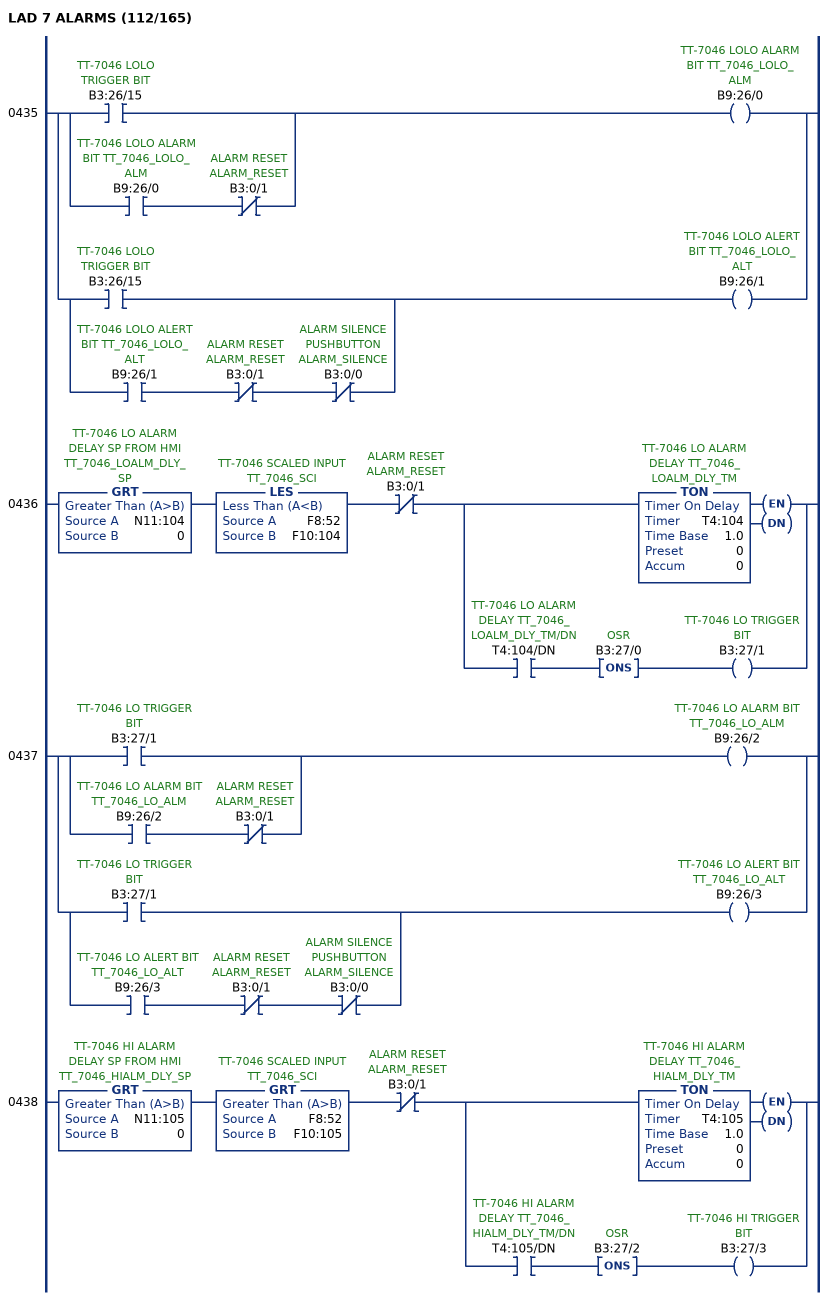
% Rung: 435 %
SOR BST BST XIC B3:26/15 NXB XIC B9:26/0 XIO B3:0/1 BND OTE B9:26/0 NXB BST XIC B3:26/15 NXB XIC B9:26/1 XIO B3:0/1 XIO B3:0/0 BND OTE B9:26/1 BND EOR
%   B3:26/15  "TT-7046 LOLO TRIGGER BIT" %
%   B9:26/0  TT_7046_LOLO_ALM  "TT-7046 LOLO ALARM BIT" %
%   B3:0/1  ALARM_RESET  "ALARM RESET" %
%   B9:26/1  TT_7046_LOLO_ALT  "TT-7046 LOLO ALERT BIT" %
%   B3:0/0  ALARM_SILENCE  "ALARM SILENCE PUSHBUTTON" %
% Rung: 436 %
SOR GRT N11:104 0 LES F8:52 F10:104 XIO B3:0/1 BST TON T4:104 1.0 0 0 NXB XIC T4:104/DN OSR B3:27/0 OTE B3:27/1 BND EOR
%   N11:104  TT_7046_LOALM_DLY_SP  "TT-7046 LO ALARM DELAY SP FROM HMI" %
%   F8:52  TT_7046_SCI  "TT-7046 SCALED INPUT" %
%   F10:104  TT_7046_LOALM_SP  "TT-7046 LO ALARM SP" %
%   B3:0/1  ALARM_RESET  "ALARM RESET" %
%   T4:104  TT_7046_LOALM_DLY_TM  "TT-7046 LO ALARM DELAY" %
%   B3:27/0  "OSR" %
%   B3:27/1  "TT-7046 LO TRIGGER BIT" %
% Rung: 437 %
SOR BST BST XIC B3:27/1 NXB XIC B9:26/2 XIO B3:0/1 BND OTE B9:26/2 NXB BST XIC B3:27/1 NXB XIC B9:26/3 XIO B3:0/1 XIO B3:0/0 BND OTE B9:26/3 BND EOR
%   B3:27/1  "TT-7046 LO TRIGGER BIT" %
%   B9:26/2  TT_7046_LO_ALM  "TT-7046 LO ALARM BIT" %
%   B3:0/1  ALARM_RESET  "ALARM RESET" %
%   B9:26/3  TT_7046_LO_ALT  "TT-7046 LO ALERT BIT" %
%   B3:0/0  ALARM_SILENCE  "ALARM SILENCE PUSHBUTTON" %
% Rung: 438 %
SOR GRT N11:105 0 GRT F8:52 F10:105 XIO B3:0/1 BST TON T4:105 1.0 0 0 NXB XIC T4:105/DN OSR B3:27/2 OTE B3:27/3 BND EOR
%   N11:105  TT_7046_HIALM_DLY_SP  "TT-7046 HI ALARM DELAY SP FROM HMI" %
%   F8:52  TT_7046_SCI  "TT-7046 SCALED INPUT" %
%   F10:105  TT_7046_HIALM_SP  "TT-7046 HI ALARM SP" %
%   B3:0/1  ALARM_RESET  "ALARM RESET" %
%   T4:105  TT_7046_HIALM_DLY_TM  "TT-7046 HI ALARM DELAY" %
%   B3:27/2  "OSR" %
%   B3:27/3  "TT-7046 HI TRIGGER BIT" %

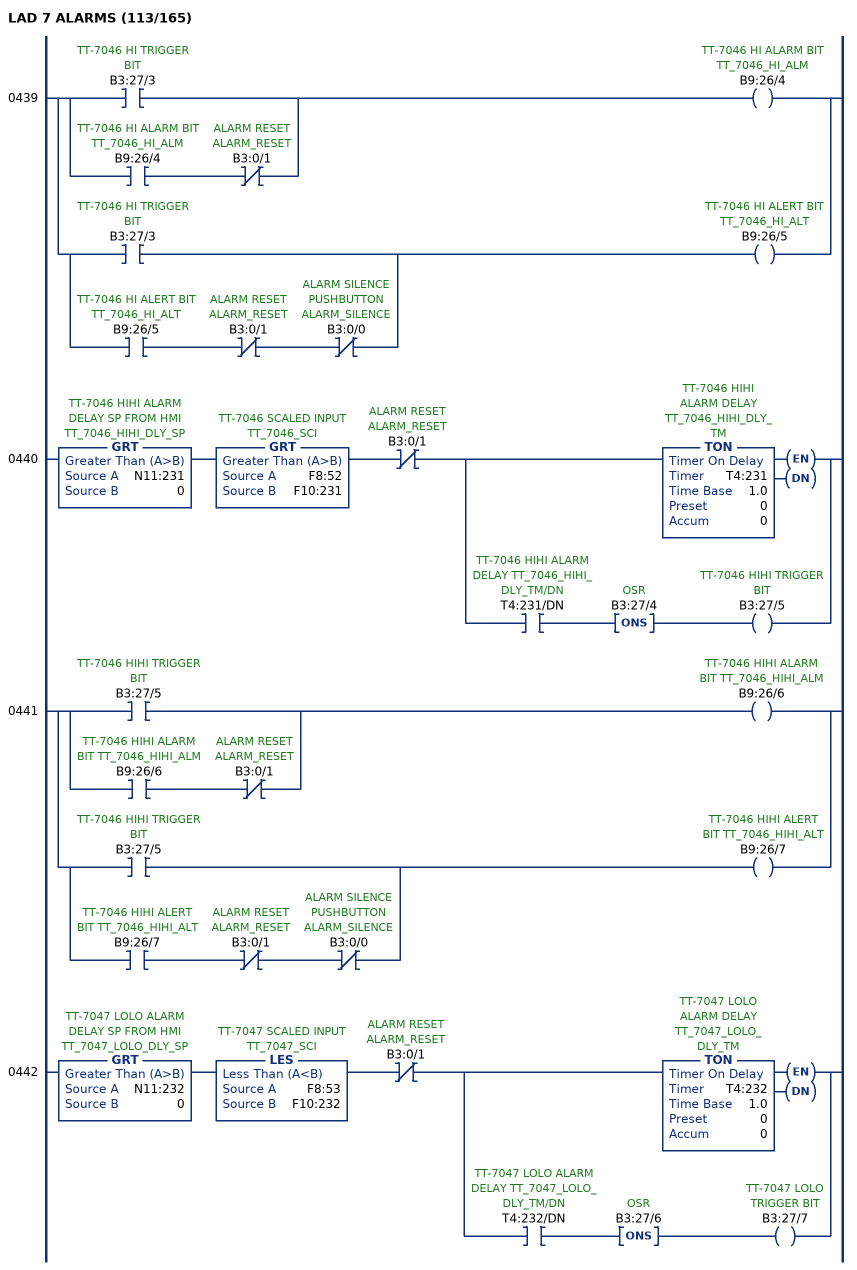
% Rung: 439 %
SOR BST BST XIC B3:27/3 NXB XIC B9:26/4 XIO B3:0/1 BND OTE B9:26/4 NXB BST XIC B3:27/3 NXB XIC B9:26/5 XIO B3:0/1 XIO B3:0/0 BND OTE B9:26/5 BND EOR
%   B3:27/3  "TT-7046 HI TRIGGER BIT" %
%   B9:26/4  TT_7046_HI_ALM  "TT-7046 HI ALARM BIT" %
%   B3:0/1  ALARM_RESET  "ALARM RESET" %
%   B9:26/5  TT_7046_HI_ALT  "TT-7046 HI ALERT BIT" %
%   B3:0/0  ALARM_SILENCE  "ALARM SILENCE PUSHBUTTON" %
% Rung: 440 %
SOR GRT N11:231 0 GRT F8:52 F10:231 XIO B3:0/1 BST TON T4:231 1.0 0 0 NXB XIC T4:231/DN OSR B3:27/4 OTE B3:27/5 BND EOR
%   N11:231  TT_7046_HIHI_DLY_SP  "TT-7046 HIHI ALARM DELAY SP FROM HMI" %
%   F8:52  TT_7046_SCI  "TT-7046 SCALED INPUT" %
%   F10:231  TT_7046_HIHI_SP  "TT-7046 HIHI ALARM SP" %
%   B3:0/1  ALARM_RESET  "ALARM RESET" %
%   T4:231  TT_7046_HIHI_DLY_TM  "TT-7046 HIHI ALARM DELAY" %
%   B3:27/4  "OSR" %
%   B3:27/5  "TT-7046 HIHI TRIGGER BIT" %
% Rung: 441 %
SOR BST BST XIC B3:27/5 NXB XIC B9:26/6 XIO B3:0/1 BND OTE B9:26/6 NXB BST XIC B3:27/5 NXB XIC B9:26/7 XIO B3:0/1 XIO B3:0/0 BND OTE B9:26/7 BND EOR
%   B3:27/5  "TT-7046 HIHI TRIGGER BIT" %
%   B9:26/6  TT_7046_HIHI_ALM  "TT-7046 HIHI ALARM BIT" %
%   B3:0/1  ALARM_RESET  "ALARM RESET" %
%   B9:26/7  TT_7046_HIHI_ALT  "TT-7046 HIHI ALERT BIT" %
%   B3:0/0  ALARM_SILENCE  "ALARM SILENCE PUSHBUTTON" %
% Rung: 442 %
SOR GRT N11:232 0 LES F8:53 F10:232 XIO B3:0/1 BST TON T4:232 1.0 0 0 NXB XIC T4:232/DN OSR B3:27/6 OTE B3:27/7 BND EOR
%   N11:232  TT_7047_LOLO_DLY_SP  "TT-7047 LOLO ALARM DELAY SP FROM HMI" %
%   F8:53  TT_7047_SCI  "TT-7047 SCALED INPUT" %
%   F10:232  TT_7047_LOLO_SP  "TT-7047 LOLO ALARM SP" %
%   B3:0/1  ALARM_RESET  "ALARM RESET" %
%   T4:232  TT_7047_LOLO_DLY_TM  "TT-7047 LOLO ALARM DELAY" %
%   B3:27/6  "OSR" %
%   B3:27/7  "TT-7047 LOLO TRIGGER BIT" %

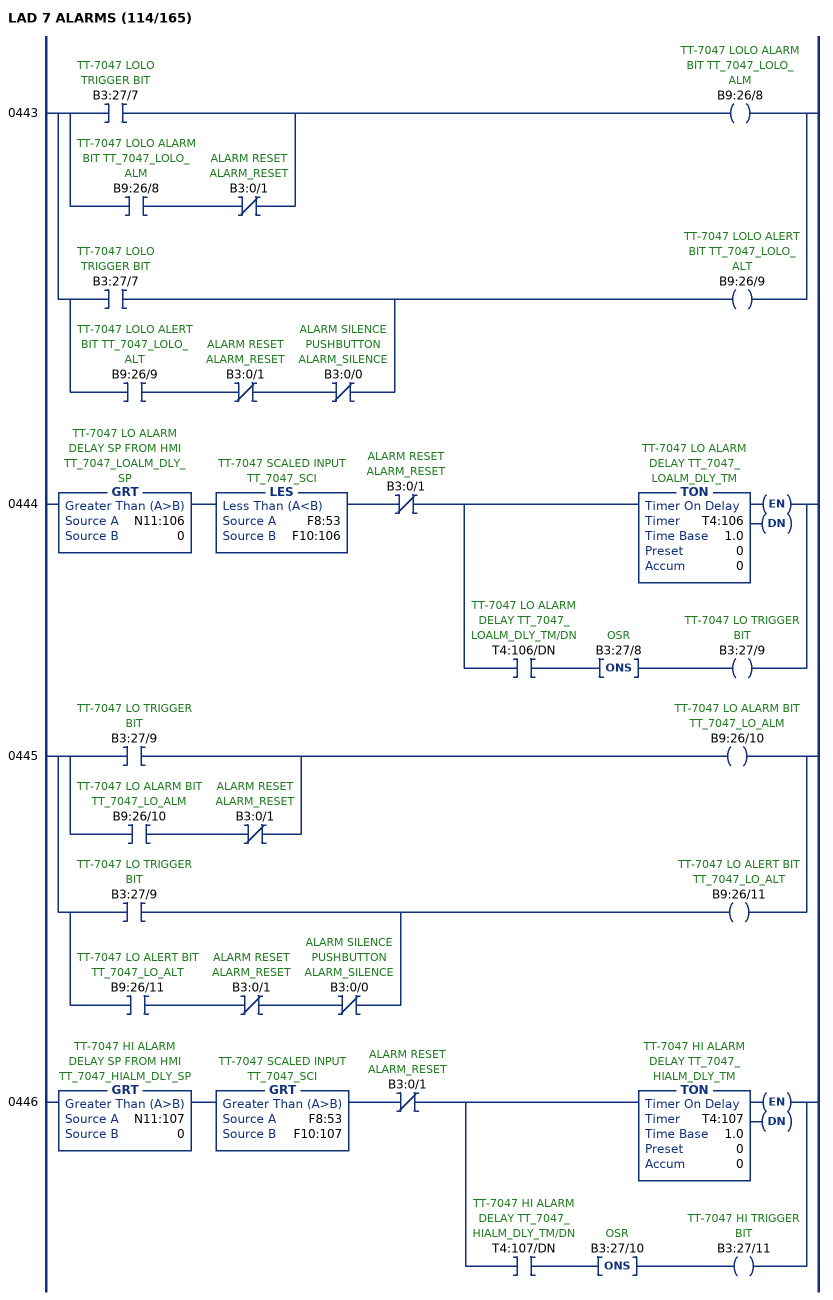
% Rung: 443 %
SOR BST BST XIC B3:27/7 NXB XIC B9:26/8 XIO B3:0/1 BND OTE B9:26/8 NXB BST XIC B3:27/7 NXB XIC B9:26/9 XIO B3:0/1 XIO B3:0/0 BND OTE B9:26/9 BND EOR
%   B3:27/7  "TT-7047 LOLO TRIGGER BIT" %
%   B9:26/8  TT_7047_LOLO_ALM  "TT-7047 LOLO ALARM BIT" %
%   B3:0/1  ALARM_RESET  "ALARM RESET" %
%   B9:26/9  TT_7047_LOLO_ALT  "TT-7047 LOLO ALERT BIT" %
%   B3:0/0  ALARM_SILENCE  "ALARM SILENCE PUSHBUTTON" %
% Rung: 444 %
SOR GRT N11:106 0 LES F8:53 F10:106 XIO B3:0/1 BST TON T4:106 1.0 0 0 NXB XIC T4:106/DN OSR B3:27/8 OTE B3:27/9 BND EOR
%   N11:106  TT_7047_LOALM_DLY_SP  "TT-7047 LO ALARM DELAY SP FROM HMI" %
%   F8:53  TT_7047_SCI  "TT-7047 SCALED INPUT" %
%   F10:106  TT_7047_LOALM_SP  "TT-7047 LO ALARM SP" %
%   B3:0/1  ALARM_RESET  "ALARM RESET" %
%   T4:106  TT_7047_LOALM_DLY_TM  "TT-7047 LO ALARM DELAY" %
%   B3:27/8  "OSR" %
%   B3:27/9  "TT-7047 LO TRIGGER BIT" %
% Rung: 445 %
SOR BST BST XIC B3:27/9 NXB XIC B9:26/10 XIO B3:0/1 BND OTE B9:26/10 NXB BST XIC B3:27/9 NXB XIC B9:26/11 XIO B3:0/1 XIO B3:0/0 BND OTE B9:26/11 BND EOR
%   B3:27/9  "TT-7047 LO TRIGGER BIT" %
%   B9:26/10  TT_7047_LO_ALM  "TT-7047 LO ALARM BIT" %
%   B3:0/1  ALARM_RESET  "ALARM RESET" %
%   B9:26/11  TT_7047_LO_ALT  "TT-7047 LO ALERT BIT" %
%   B3:0/0  ALARM_SILENCE  "ALARM SILENCE PUSHBUTTON" %
% Rung: 446 %
SOR GRT N11:107 0 GRT F8:53 F10:107 XIO B3:0/1 BST TON T4:107 1.0 0 0 NXB XIC T4:107/DN OSR B3:27/10 OTE B3:27/11 BND EOR
%   N11:107  TT_7047_HIALM_DLY_SP  "TT-7047 HI ALARM DELAY SP FROM HMI" %
%   F8:53  TT_7047_SCI  "TT-7047 SCALED INPUT" %
%   F10:107  TT_7047_HIALM_SP  "TT-7047 HI ALARM SP" %
%   B3:0/1  ALARM_RESET  "ALARM RESET" %
%   T4:107  TT_7047_HIALM_DLY_TM  "TT-7047 HI ALARM DELAY" %
%   B3:27/10  "OSR" %
%   B3:27/11  "TT-7047 HI TRIGGER BIT" %

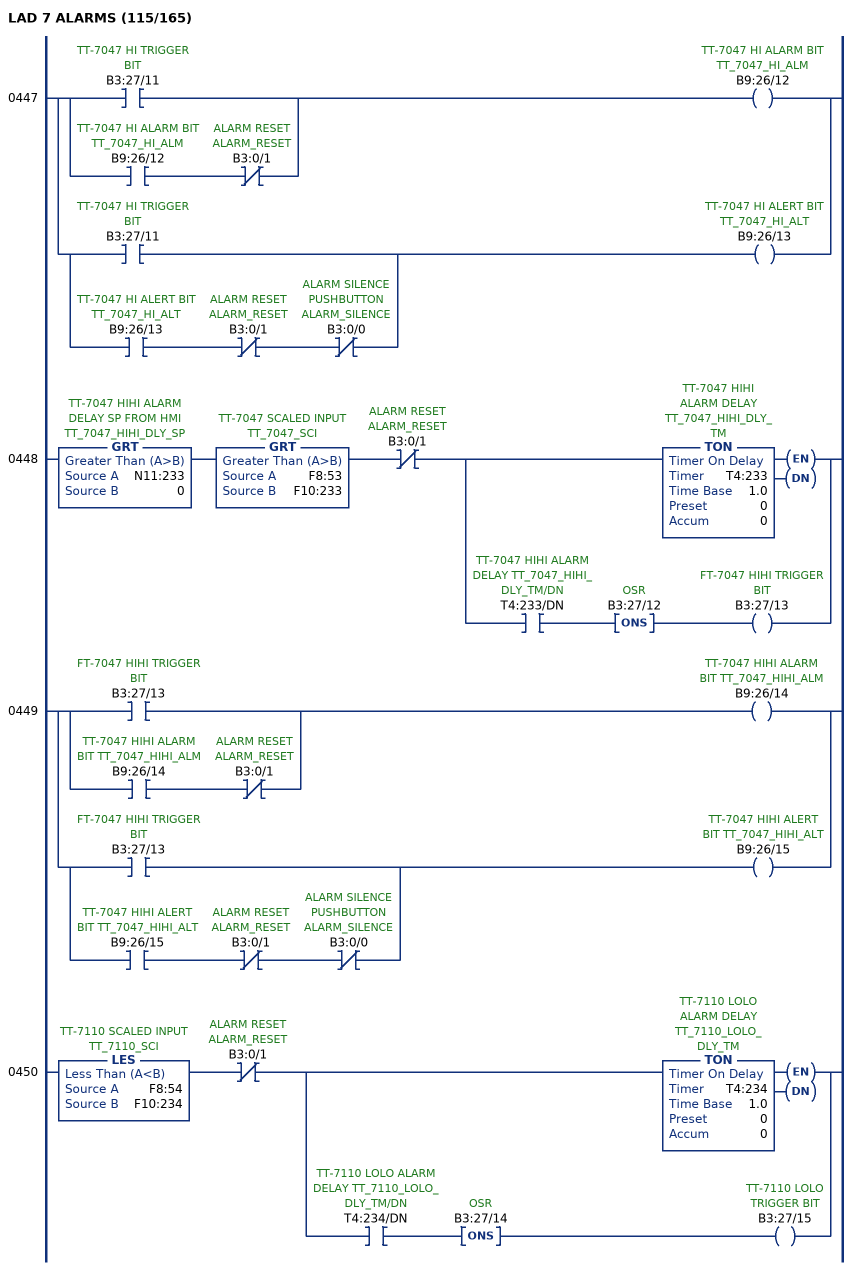
% Rung: 447 %
SOR BST BST XIC B3:27/11 NXB XIC B9:26/12 XIO B3:0/1 BND OTE B9:26/12 NXB BST XIC B3:27/11 NXB XIC B9:26/13 XIO B3:0/1 XIO B3:0/0 BND OTE B9:26/13 BND EOR
%   B3:27/11  "TT-7047 HI TRIGGER BIT" %
%   B9:26/12  TT_7047_HI_ALM  "TT-7047 HI ALARM BIT" %
%   B3:0/1  ALARM_RESET  "ALARM RESET" %
%   B9:26/13  TT_7047_HI_ALT  "TT-7047 HI ALERT BIT" %
%   B3:0/0  ALARM_SILENCE  "ALARM SILENCE PUSHBUTTON" %
% Rung: 448 %
SOR GRT N11:233 0 GRT F8:53 F10:233 XIO B3:0/1 BST TON T4:233 1.0 0 0 NXB XIC T4:233/DN OSR B3:27/12 OTE B3:27/13 BND EOR
%   N11:233  TT_7047_HIHI_DLY_SP  "TT-7047 HIHI ALARM DELAY SP FROM HMI" %
%   F8:53  TT_7047_SCI  "TT-7047 SCALED INPUT" %
%   F10:233  TT_7047_HIHI_SP  "TT-7047 HIHI ALARM SP" %
%   B3:0/1  ALARM_RESET  "ALARM RESET" %
%   T4:233  TT_7047_HIHI_DLY_TM  "TT-7047 HIHI ALARM DELAY" %
%   B3:27/12  "OSR" %
%   B3:27/13  "FT-7047 HIHI TRIGGER BIT" %
% Rung: 449 %
SOR BST BST XIC B3:27/13 NXB XIC B9:26/14 XIO B3:0/1 BND OTE B9:26/14 NXB BST XIC B3:27/13 NXB XIC B9:26/15 XIO B3:0/1 XIO B3:0/0 BND OTE B9:26/15 BND EOR
%   B3:27/13  "FT-7047 HIHI TRIGGER BIT" %
%   B9:26/14  TT_7047_HIHI_ALM  "TT-7047 HIHI ALARM BIT" %
%   B3:0/1  ALARM_RESET  "ALARM RESET" %
%   B9:26/15  TT_7047_HIHI_ALT  "TT-7047 HIHI ALERT BIT" %
%   B3:0/0  ALARM_SILENCE  "ALARM SILENCE PUSHBUTTON" %
% Rung: 450 %
SOR LES F8:54 F10:234 XIO B3:0/1 BST TON T4:234 1.0 0 0 NXB XIC T4:234/DN OSR B3:27/14 OTE B3:27/15 BND EOR
%   F8:54  TT_7110_SCI  "TT-7110 SCALED INPUT" %
%   F10:234  TT_7110_LOLO_SP  "TT-7110 LOLO ALARM SP" %
%   B3:0/1  ALARM_RESET  "ALARM RESET" %
%   T4:234  TT_7110_LOLO_DLY_TM  "TT-7110 LOLO ALARM DELAY" %
%   B3:27/14  "OSR" %
%   B3:27/15  "TT-7110 LOLO TRIGGER BIT" %

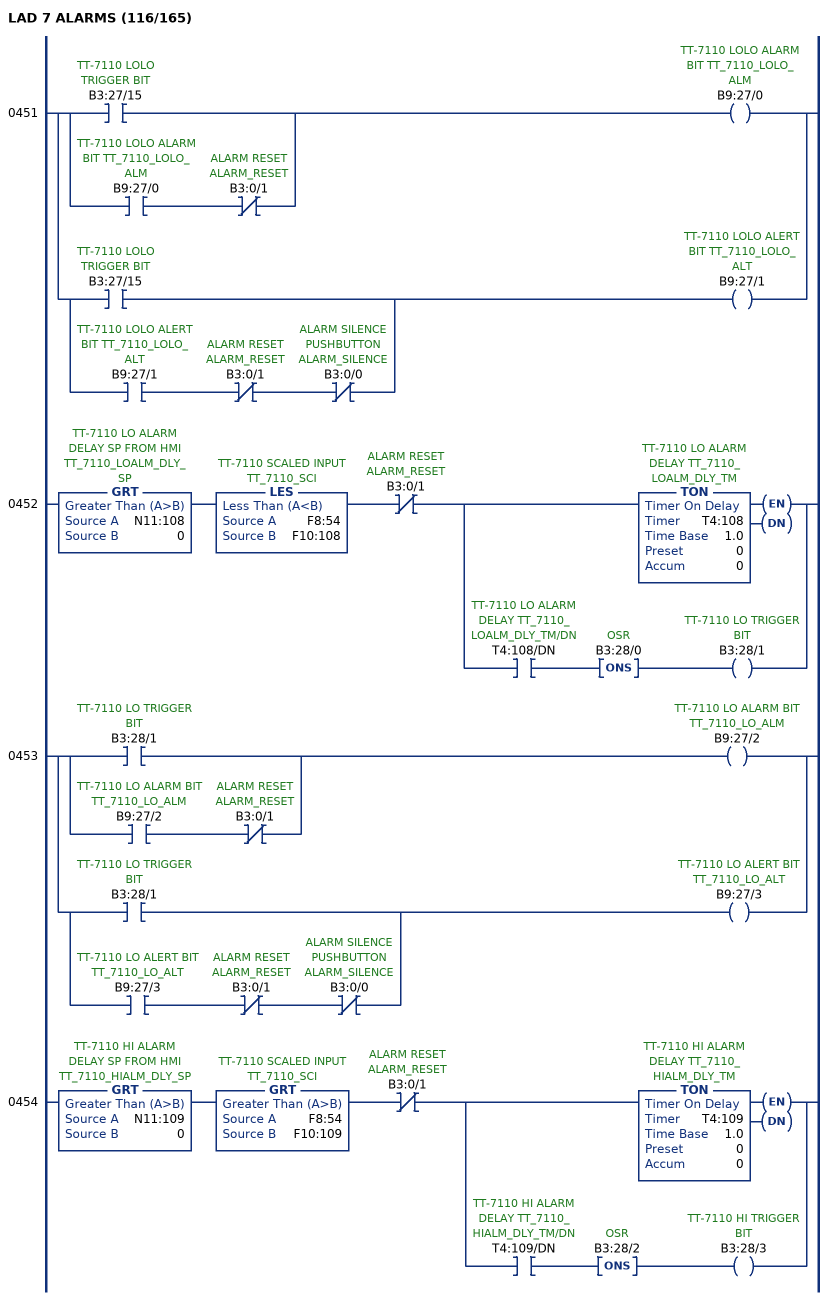
% Rung: 451 %
SOR BST BST XIC B3:27/15 NXB XIC B9:27/0 XIO B3:0/1 BND OTE B9:27/0 NXB BST XIC B3:27/15 NXB XIC B9:27/1 XIO B3:0/1 XIO B3:0/0 BND OTE B9:27/1 BND EOR
%   B3:27/15  "TT-7110 LOLO TRIGGER BIT" %
%   B9:27/0  TT_7110_LOLO_ALM  "TT-7110 LOLO ALARM BIT" %
%   B3:0/1  ALARM_RESET  "ALARM RESET" %
%   B9:27/1  TT_7110_LOLO_ALT  "TT-7110 LOLO ALERT BIT" %
%   B3:0/0  ALARM_SILENCE  "ALARM SILENCE PUSHBUTTON" %
% Rung: 452 %
SOR GRT N11:108 0 LES F8:54 F10:108 XIO B3:0/1 BST TON T4:108 1.0 0 0 NXB XIC T4:108/DN OSR B3:28/0 OTE B3:28/1 BND EOR
%   N11:108  TT_7110_LOALM_DLY_SP  "TT-7110 LO ALARM DELAY SP FROM HMI" %
%   F8:54  TT_7110_SCI  "TT-7110 SCALED INPUT" %
%   F10:108  TT_7110_LOALM_SP  "TT-7110 LO ALARM SP" %
%   B3:0/1  ALARM_RESET  "ALARM RESET" %
%   T4:108  TT_7110_LOALM_DLY_TM  "TT-7110 LO ALARM DELAY" %
%   B3:28/0  "OSR" %
%   B3:28/1  "TT-7110 LO TRIGGER BIT" %
% Rung: 453 %
SOR BST BST XIC B3:28/1 NXB XIC B9:27/2 XIO B3:0/1 BND OTE B9:27/2 NXB BST XIC B3:28/1 NXB XIC B9:27/3 XIO B3:0/1 XIO B3:0/0 BND OTE B9:27/3 BND EOR
%   B3:28/1  "TT-7110 LO TRIGGER BIT" %
%   B9:27/2  TT_7110_LO_ALM  "TT-7110 LO ALARM BIT" %
%   B3:0/1  ALARM_RESET  "ALARM RESET" %
%   B9:27/3  TT_7110_LO_ALT  "TT-7110 LO ALERT BIT" %
%   B3:0/0  ALARM_SILENCE  "ALARM SILENCE PUSHBUTTON" %
% Rung: 454 %
SOR GRT N11:109 0 GRT F8:54 F10:109 XIO B3:0/1 BST TON T4:109 1.0 0 0 NXB XIC T4:109/DN OSR B3:28/2 OTE B3:28/3 BND EOR
%   N11:109  TT_7110_HIALM_DLY_SP  "TT-7110 HI ALARM DELAY SP FROM HMI" %
%   F8:54  TT_7110_SCI  "TT-7110 SCALED INPUT" %
%   F10:109  TT_7110_HIALM_SP  "TT-7110 HI ALARM SP" %
%   B3:0/1  ALARM_RESET  "ALARM RESET" %
%   T4:109  TT_7110_HIALM_DLY_TM  "TT-7110 HI ALARM DELAY" %
%   B3:28/2  "OSR" %
%   B3:28/3  "TT-7110 HI TRIGGER BIT" %

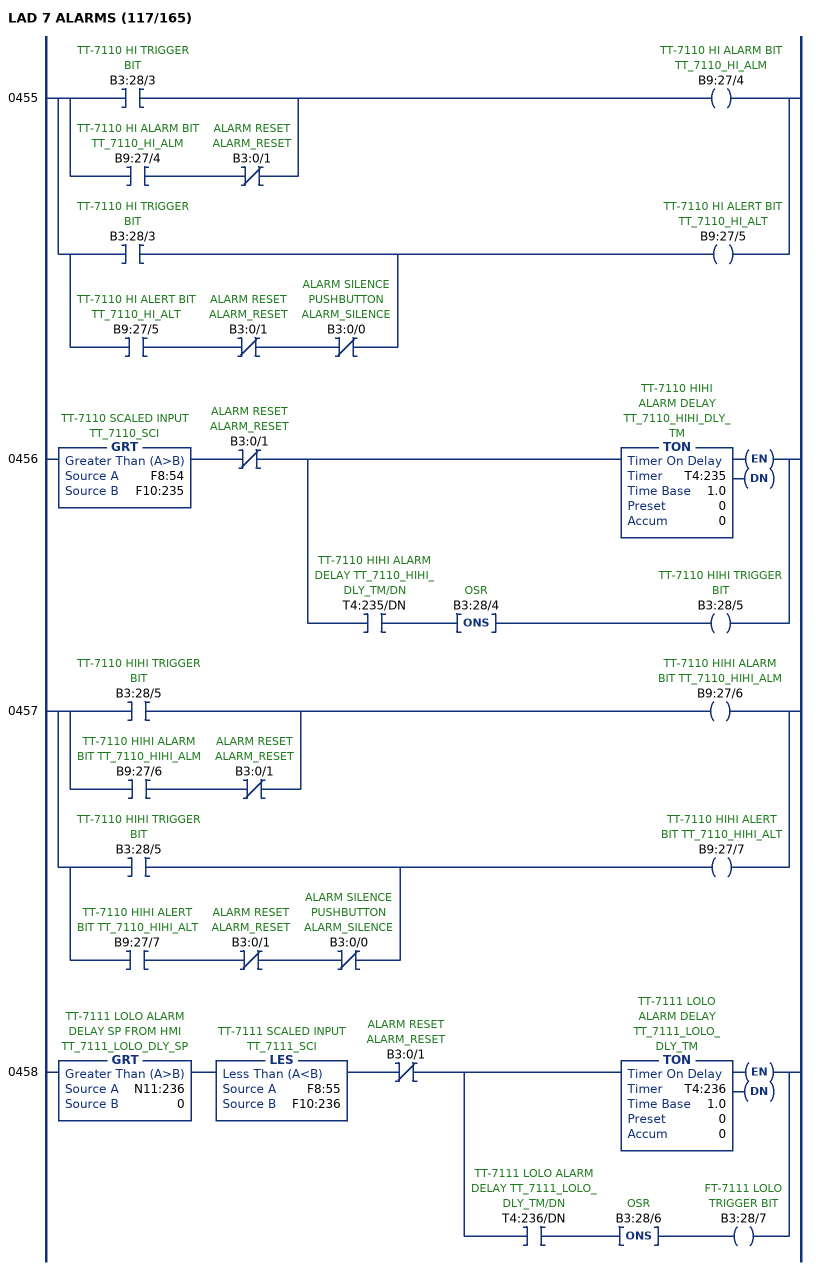
% Rung: 455 %
SOR BST BST XIC B3:28/3 NXB XIC B9:27/4 XIO B3:0/1 BND OTE B9:27/4 NXB BST XIC B3:28/3 NXB XIC B9:27/5 XIO B3:0/1 XIO B3:0/0 BND OTE B9:27/5 BND EOR
%   B3:28/3  "TT-7110 HI TRIGGER BIT" %
%   B9:27/4  TT_7110_HI_ALM  "TT-7110 HI ALARM BIT" %
%   B3:0/1  ALARM_RESET  "ALARM RESET" %
%   B9:27/5  TT_7110_HI_ALT  "TT-7110 HI ALERT BIT" %
%   B3:0/0  ALARM_SILENCE  "ALARM SILENCE PUSHBUTTON" %
% Rung: 456 %
SOR GRT F8:54 F10:235 XIO B3:0/1 BST TON T4:235 1.0 0 0 NXB XIC T4:235/DN OSR B3:28/4 OTE B3:28/5 BND EOR
%   F8:54  TT_7110_SCI  "TT-7110 SCALED INPUT" %
%   F10:235  TT_7110_HIHI_SP  "TT-7110 HIHI ALARM SP" %
%   B3:0/1  ALARM_RESET  "ALARM RESET" %
%   T4:235  TT_7110_HIHI_DLY_TM  "TT-7110 HIHI ALARM DELAY" %
%   B3:28/4  "OSR" %
%   B3:28/5  "TT-7110 HIHI TRIGGER BIT" %
% Rung: 457 %
SOR BST BST XIC B3:28/5 NXB XIC B9:27/6 XIO B3:0/1 BND OTE B9:27/6 NXB BST XIC B3:28/5 NXB XIC B9:27/7 XIO B3:0/1 XIO B3:0/0 BND OTE B9:27/7 BND EOR
%   B3:28/5  "TT-7110 HIHI TRIGGER BIT" %
%   B9:27/6  TT_7110_HIHI_ALM  "TT-7110 HIHI ALARM BIT" %
%   B3:0/1  ALARM_RESET  "ALARM RESET" %
%   B9:27/7  TT_7110_HIHI_ALT  "TT-7110 HIHI ALERT BIT" %
%   B3:0/0  ALARM_SILENCE  "ALARM SILENCE PUSHBUTTON" %
% Rung: 458 %
SOR GRT N11:236 0 LES F8:55 F10:236 XIO B3:0/1 BST TON T4:236 1.0 0 0 NXB XIC T4:236/DN OSR B3:28/6 OTE B3:28/7 BND EOR
%   N11:236  TT_7111_LOLO_DLY_SP  "TT-7111 LOLO ALARM DELAY SP FROM HMI" %
%   F8:55  TT_7111_SCI  "TT-7111 SCALED INPUT" %
%   F10:236  TT_7111_LOLO_SP  "TT-7111 LOLO ALARM SP" %
%   B3:0/1  ALARM_RESET  "ALARM RESET" %
%   T4:236  TT_7111_LOLO_DLY_TM  "TT-7111 LOLO ALARM DELAY" %
%   B3:28/6  "OSR" %
%   B3:28/7  "FT-7111 LOLO TRIGGER BIT" %

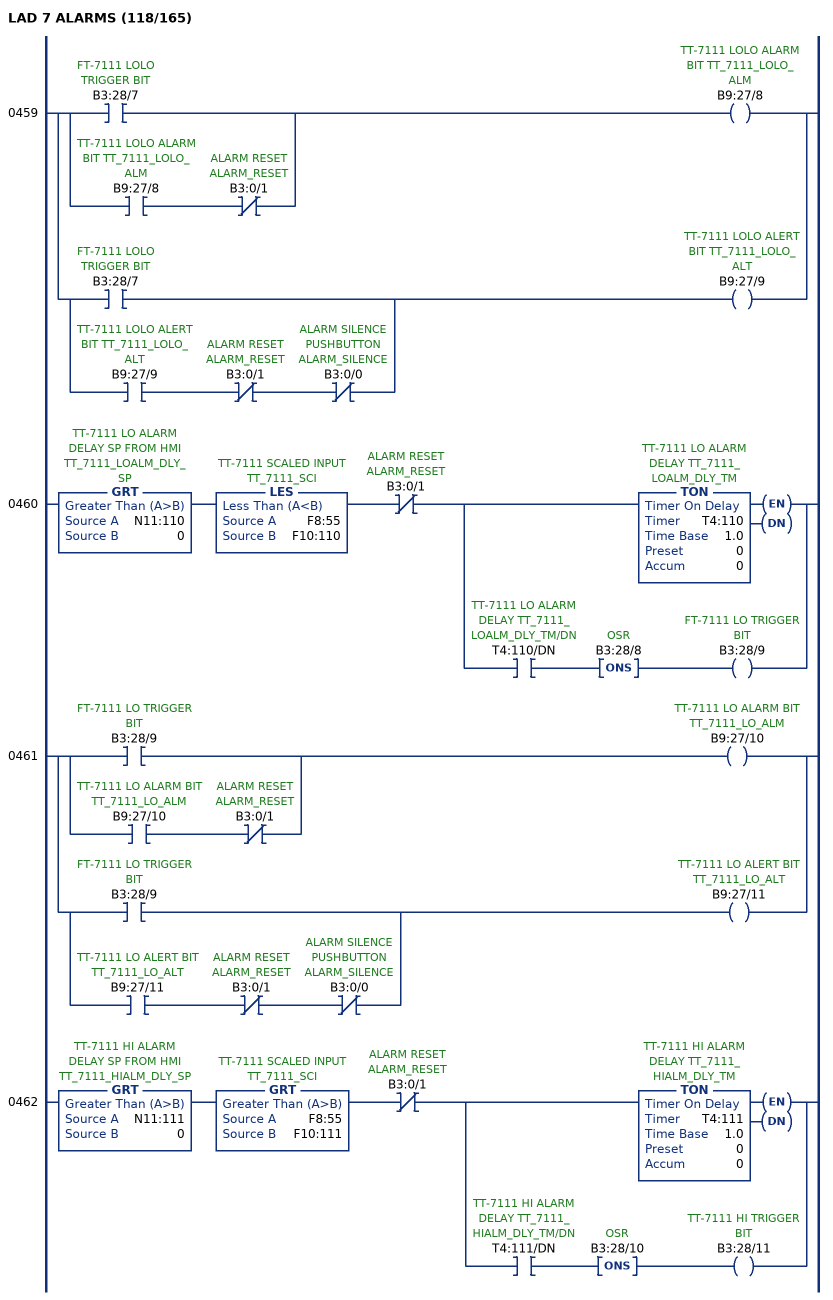
% Rung: 459 %
SOR BST BST XIC B3:28/7 NXB XIC B9:27/8 XIO B3:0/1 BND OTE B9:27/8 NXB BST XIC B3:28/7 NXB XIC B9:27/9 XIO B3:0/1 XIO B3:0/0 BND OTE B9:27/9 BND EOR
%   B3:28/7  "FT-7111 LOLO TRIGGER BIT" %
%   B9:27/8  TT_7111_LOLO_ALM  "TT-7111 LOLO ALARM BIT" %
%   B3:0/1  ALARM_RESET  "ALARM RESET" %
%   B9:27/9  TT_7111_LOLO_ALT  "TT-7111 LOLO ALERT BIT" %
%   B3:0/0  ALARM_SILENCE  "ALARM SILENCE PUSHBUTTON" %
% Rung: 460 %
SOR GRT N11:110 0 LES F8:55 F10:110 XIO B3:0/1 BST TON T4:110 1.0 0 0 NXB XIC T4:110/DN OSR B3:28/8 OTE B3:28/9 BND EOR
%   N11:110  TT_7111_LOALM_DLY_SP  "TT-7111 LO ALARM DELAY SP FROM HMI" %
%   F8:55  TT_7111_SCI  "TT-7111 SCALED INPUT" %
%   F10:110  TT_7111_LOALM_SP  "TT-7111 LO ALARM SP" %
%   B3:0/1  ALARM_RESET  "ALARM RESET" %
%   T4:110  TT_7111_LOALM_DLY_TM  "TT-7111 LO ALARM DELAY" %
%   B3:28/8  "OSR" %
%   B3:28/9  "FT-7111 LO TRIGGER BIT" %
% Rung: 461 %
SOR BST BST XIC B3:28/9 NXB XIC B9:27/10 XIO B3:0/1 BND OTE B9:27/10 NXB BST XIC B3:28/9 NXB XIC B9:27/11 XIO B3:0/1 XIO B3:0/0 BND OTE B9:27/11 BND EOR
%   B3:28/9  "FT-7111 LO TRIGGER BIT" %
%   B9:27/10  TT_7111_LO_ALM  "TT-7111 LO ALARM BIT" %
%   B3:0/1  ALARM_RESET  "ALARM RESET" %
%   B9:27/11  TT_7111_LO_ALT  "TT-7111 LO ALERT BIT" %
%   B3:0/0  ALARM_SILENCE  "ALARM SILENCE PUSHBUTTON" %
% Rung: 462 %
SOR GRT N11:111 0 GRT F8:55 F10:111 XIO B3:0/1 BST TON T4:111 1.0 0 0 NXB XIC T4:111/DN OSR B3:28/10 OTE B3:28/11 BND EOR
%   N11:111  TT_7111_HIALM_DLY_SP  "TT-7111 HI ALARM DELAY SP FROM HMI" %
%   F8:55  TT_7111_SCI  "TT-7111 SCALED INPUT" %
%   F10:111  TT_7111_HIALM_SP  "TT-7111 HI ALARM SP" %
%   B3:0/1  ALARM_RESET  "ALARM RESET" %
%   T4:111  TT_7111_HIALM_DLY_TM  "TT-7111 HI ALARM DELAY" %
%   B3:28/10  "OSR" %
%   B3:28/11  "TT-7111 HI TRIGGER BIT" %

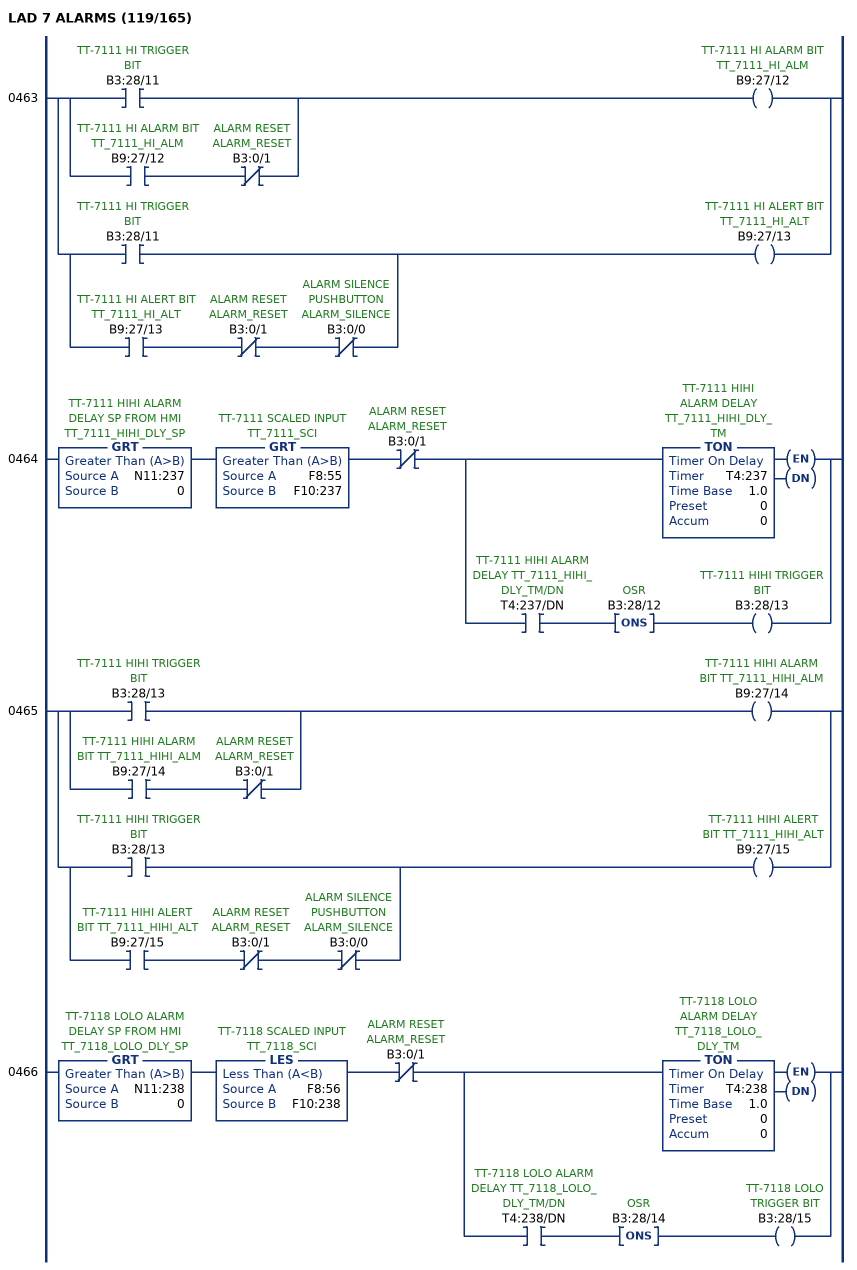
% Rung: 463 %
SOR BST BST XIC B3:28/11 NXB XIC B9:27/12 XIO B3:0/1 BND OTE B9:27/12 NXB BST XIC B3:28/11 NXB XIC B9:27/13 XIO B3:0/1 XIO B3:0/0 BND OTE B9:27/13 BND EOR
%   B3:28/11  "TT-7111 HI TRIGGER BIT" %
%   B9:27/12  TT_7111_HI_ALM  "TT-7111 HI ALARM BIT" %
%   B3:0/1  ALARM_RESET  "ALARM RESET" %
%   B9:27/13  TT_7111_HI_ALT  "TT-7111 HI ALERT BIT" %
%   B3:0/0  ALARM_SILENCE  "ALARM SILENCE PUSHBUTTON" %
% Rung: 464 %
SOR GRT N11:237 0 GRT F8:55 F10:237 XIO B3:0/1 BST TON T4:237 1.0 0 0 NXB XIC T4:237/DN OSR B3:28/12 OTE B3:28/13 BND EOR
%   N11:237  TT_7111_HIHI_DLY_SP  "TT-7111 HIHI ALARM DELAY SP FROM HMI" %
%   F8:55  TT_7111_SCI  "TT-7111 SCALED INPUT" %
%   F10:237  TT_7111_HIHI_SP  "TT-7111 HIHI ALARM SP" %
%   B3:0/1  ALARM_RESET  "ALARM RESET" %
%   T4:237  TT_7111_HIHI_DLY_TM  "TT-7111 HIHI ALARM DELAY" %
%   B3:28/12  "OSR" %
%   B3:28/13  "TT-7111 HIHI TRIGGER BIT" %
% Rung: 465 %
SOR BST BST XIC B3:28/13 NXB XIC B9:27/14 XIO B3:0/1 BND OTE B9:27/14 NXB BST XIC B3:28/13 NXB XIC B9:27/15 XIO B3:0/1 XIO B3:0/0 BND OTE B9:27/15 BND EOR
%   B3:28/13  "TT-7111 HIHI TRIGGER BIT" %
%   B9:27/14  TT_7111_HIHI_ALM  "TT-7111 HIHI ALARM BIT" %
%   B3:0/1  ALARM_RESET  "ALARM RESET" %
%   B9:27/15  TT_7111_HIHI_ALT  "TT-7111 HIHI ALERT BIT" %
%   B3:0/0  ALARM_SILENCE  "ALARM SILENCE PUSHBUTTON" %
% Rung: 466 %
SOR GRT N11:238 0 LES F8:56 F10:238 XIO B3:0/1 BST TON T4:238 1.0 0 0 NXB XIC T4:238/DN OSR B3:28/14 OTE B3:28/15 BND EOR
%   N11:238  TT_7118_LOLO_DLY_SP  "TT-7118 LOLO ALARM DELAY SP FROM HMI" %
%   F8:56  TT_7118_SCI  "TT-7118 SCALED INPUT" %
%   F10:238  TT_7118_LOLO_SP  "TT-7118 LOLO ALARM SP" %
%   B3:0/1  ALARM_RESET  "ALARM RESET" %
%   T4:238  TT_7118_LOLO_DLY_TM  "TT-7118 LOLO ALARM DELAY" %
%   B3:28/14  "OSR" %
%   B3:28/15  "TT-7118 LOLO TRIGGER BIT" %

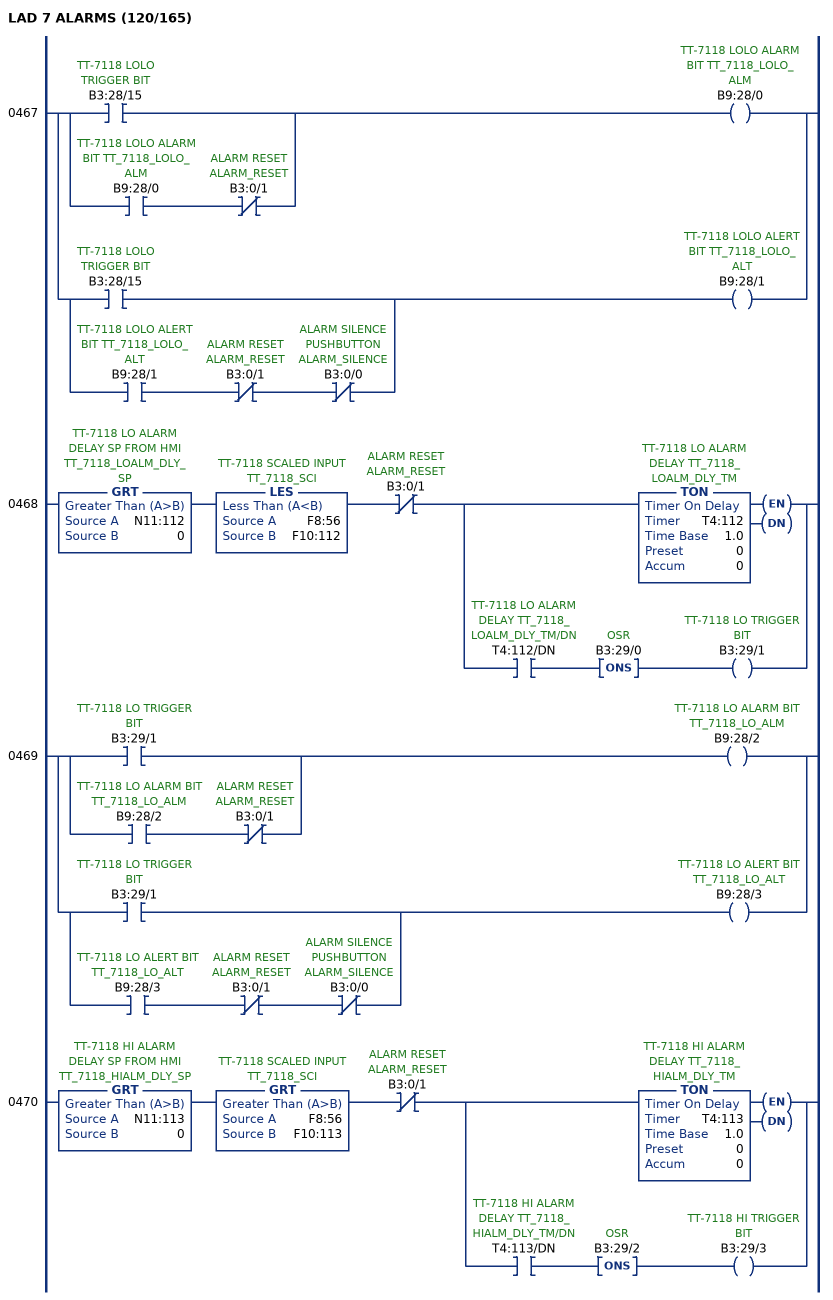
% Rung: 467 %
SOR BST BST XIC B3:28/15 NXB XIC B9:28/0 XIO B3:0/1 BND OTE B9:28/0 NXB BST XIC B3:28/15 NXB XIC B9:28/1 XIO B3:0/1 XIO B3:0/0 BND OTE B9:28/1 BND EOR
%   B3:28/15  "TT-7118 LOLO TRIGGER BIT" %
%   B9:28/0  TT_7118_LOLO_ALM  "TT-7118 LOLO ALARM BIT" %
%   B3:0/1  ALARM_RESET  "ALARM RESET" %
%   B9:28/1  TT_7118_LOLO_ALT  "TT-7118 LOLO ALERT BIT" %
%   B3:0/0  ALARM_SILENCE  "ALARM SILENCE PUSHBUTTON" %
% Rung: 468 %
SOR GRT N11:112 0 LES F8:56 F10:112 XIO B3:0/1 BST TON T4:112 1.0 0 0 NXB XIC T4:112/DN OSR B3:29/0 OTE B3:29/1 BND EOR
%   N11:112  TT_7118_LOALM_DLY_SP  "TT-7118 LO ALARM DELAY SP FROM HMI" %
%   F8:56  TT_7118_SCI  "TT-7118 SCALED INPUT" %
%   F10:112  TT_7118_LOALM_SP  "TT-7118 LO ALARM SP" %
%   B3:0/1  ALARM_RESET  "ALARM RESET" %
%   T4:112  TT_7118_LOALM_DLY_TM  "TT-7118 LO ALARM DELAY" %
%   B3:29/0  "OSR" %
%   B3:29/1  "TT-7118 LO TRIGGER BIT" %
% Rung: 469 %
SOR BST BST XIC B3:29/1 NXB XIC B9:28/2 XIO B3:0/1 BND OTE B9:28/2 NXB BST XIC B3:29/1 NXB XIC B9:28/3 XIO B3:0/1 XIO B3:0/0 BND OTE B9:28/3 BND EOR
%   B3:29/1  "TT-7118 LO TRIGGER BIT" %
%   B9:28/2  TT_7118_LO_ALM  "TT-7118 LO ALARM BIT" %
%   B3:0/1  ALARM_RESET  "ALARM RESET" %
%   B9:28/3  TT_7118_LO_ALT  "TT-7118 LO ALERT BIT" %
%   B3:0/0  ALARM_SILENCE  "ALARM SILENCE PUSHBUTTON" %
% Rung: 470 %
SOR GRT N11:113 0 GRT F8:56 F10:113 XIO B3:0/1 BST TON T4:113 1.0 0 0 NXB XIC T4:113/DN OSR B3:29/2 OTE B3:29/3 BND EOR
%   N11:113  TT_7118_HIALM_DLY_SP  "TT-7118 HI ALARM DELAY SP FROM HMI" %
%   F8:56  TT_7118_SCI  "TT-7118 SCALED INPUT" %
%   F10:113  TT_7118_HIALM_SP  "TT-7118 HI ALARM SP" %
%   B3:0/1  ALARM_RESET  "ALARM RESET" %
%   T4:113  TT_7118_HIALM_DLY_TM  "TT-7118 HI ALARM DELAY" %
%   B3:29/2  "OSR" %
%   B3:29/3  "TT-7118 HI TRIGGER BIT" %

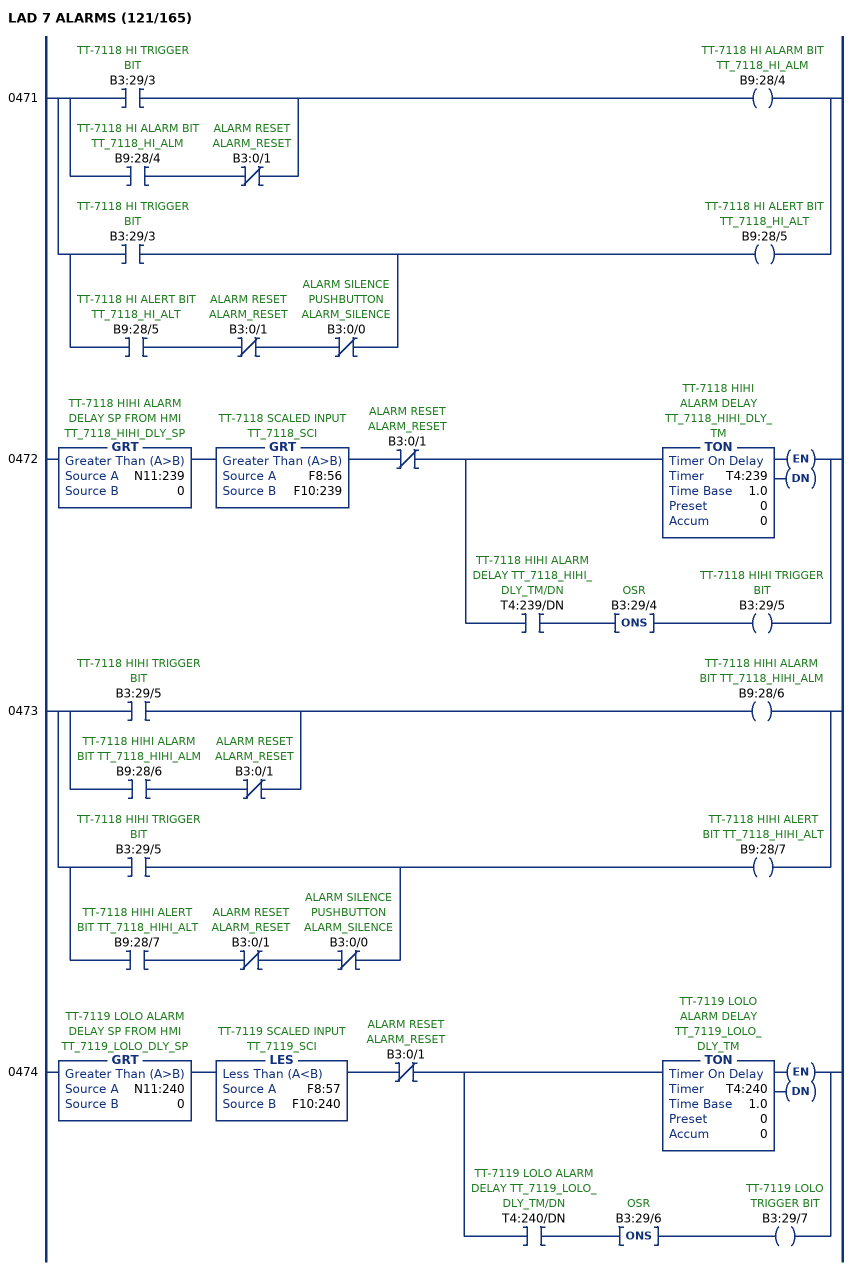
% Rung: 471 %
SOR BST BST XIC B3:29/3 NXB XIC B9:28/4 XIO B3:0/1 BND OTE B9:28/4 NXB BST XIC B3:29/3 NXB XIC B9:28/5 XIO B3:0/1 XIO B3:0/0 BND OTE B9:28/5 BND EOR
%   B3:29/3  "TT-7118 HI TRIGGER BIT" %
%   B9:28/4  TT_7118_HI_ALM  "TT-7118 HI ALARM BIT" %
%   B3:0/1  ALARM_RESET  "ALARM RESET" %
%   B9:28/5  TT_7118_HI_ALT  "TT-7118 HI ALERT BIT" %
%   B3:0/0  ALARM_SILENCE  "ALARM SILENCE PUSHBUTTON" %
% Rung: 472 %
SOR GRT N11:239 0 GRT F8:56 F10:239 XIO B3:0/1 BST TON T4:239 1.0 0 0 NXB XIC T4:239/DN OSR B3:29/4 OTE B3:29/5 BND EOR
%   N11:239  TT_7118_HIHI_DLY_SP  "TT-7118 HIHI ALARM DELAY SP FROM HMI" %
%   F8:56  TT_7118_SCI  "TT-7118 SCALED INPUT" %
%   F10:239  TT_7118_HIHI_SP  "TT-7118 HIHI ALARM SP" %
%   B3:0/1  ALARM_RESET  "ALARM RESET" %
%   T4:239  TT_7118_HIHI_DLY_TM  "TT-7118 HIHI ALARM DELAY" %
%   B3:29/4  "OSR" %
%   B3:29/5  "TT-7118 HIHI TRIGGER BIT" %
% Rung: 473 %
SOR BST BST XIC B3:29/5 NXB XIC B9:28/6 XIO B3:0/1 BND OTE B9:28/6 NXB BST XIC B3:29/5 NXB XIC B9:28/7 XIO B3:0/1 XIO B3:0/0 BND OTE B9:28/7 BND EOR
%   B3:29/5  "TT-7118 HIHI TRIGGER BIT" %
%   B9:28/6  TT_7118_HIHI_ALM  "TT-7118 HIHI ALARM BIT" %
%   B3:0/1  ALARM_RESET  "ALARM RESET" %
%   B9:28/7  TT_7118_HIHI_ALT  "TT-7118 HIHI ALERT BIT" %
%   B3:0/0  ALARM_SILENCE  "ALARM SILENCE PUSHBUTTON" %
% Rung: 474 %
SOR GRT N11:240 0 LES F8:57 F10:240 XIO B3:0/1 BST TON T4:240 1.0 0 0 NXB XIC T4:240/DN OSR B3:29/6 OTE B3:29/7 BND EOR
%   N11:240  TT_7119_LOLO_DLY_SP  "TT-7119 LOLO ALARM DELAY SP FROM HMI" %
%   F8:57  TT_7119_SCI  "TT-7119 SCALED INPUT" %
%   F10:240  TT_7119_LOLO_SP  "TT-7119 LOLO ALARM SP" %
%   B3:0/1  ALARM_RESET  "ALARM RESET" %
%   T4:240  TT_7119_LOLO_DLY_TM  "TT-7119 LOLO ALARM DELAY" %
%   B3:29/6  "OSR" %
%   B3:29/7  "TT-7119 LOLO TRIGGER BIT" %

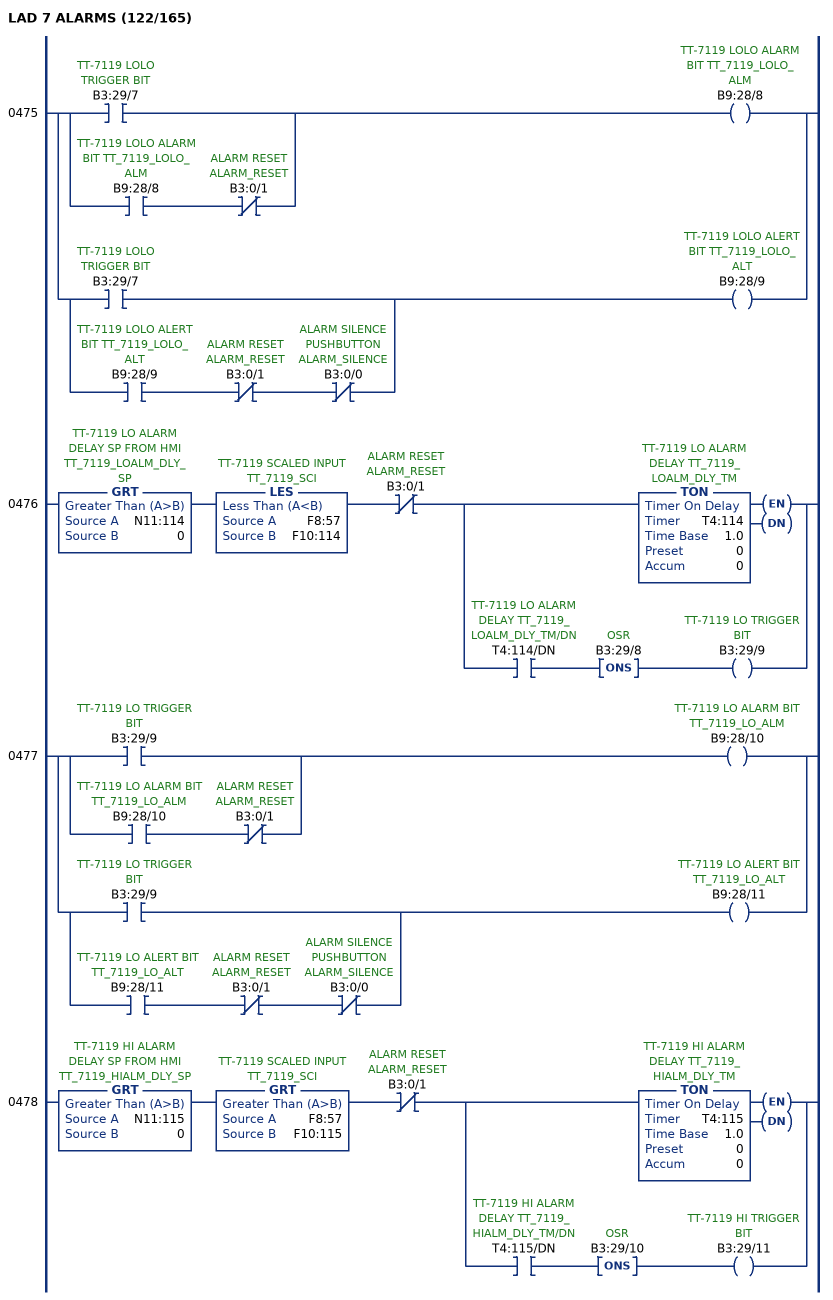
% Rung: 475 %
SOR BST BST XIC B3:29/7 NXB XIC B9:28/8 XIO B3:0/1 BND OTE B9:28/8 NXB BST XIC B3:29/7 NXB XIC B9:28/9 XIO B3:0/1 XIO B3:0/0 BND OTE B9:28/9 BND EOR
%   B3:29/7  "TT-7119 LOLO TRIGGER BIT" %
%   B9:28/8  TT_7119_LOLO_ALM  "TT-7119 LOLO ALARM BIT" %
%   B3:0/1  ALARM_RESET  "ALARM RESET" %
%   B9:28/9  TT_7119_LOLO_ALT  "TT-7119 LOLO ALERT BIT" %
%   B3:0/0  ALARM_SILENCE  "ALARM SILENCE PUSHBUTTON" %
% Rung: 476 %
SOR GRT N11:114 0 LES F8:57 F10:114 XIO B3:0/1 BST TON T4:114 1.0 0 0 NXB XIC T4:114/DN OSR B3:29/8 OTE B3:29/9 BND EOR
%   N11:114  TT_7119_LOALM_DLY_SP  "TT-7119 LO ALARM DELAY SP FROM HMI" %
%   F8:57  TT_7119_SCI  "TT-7119 SCALED INPUT" %
%   F10:114  TT_7119_LOALM_SP  "TT-7119 LO ALARM SP" %
%   B3:0/1  ALARM_RESET  "ALARM RESET" %
%   T4:114  TT_7119_LOALM_DLY_TM  "TT-7119 LO ALARM DELAY" %
%   B3:29/8  "OSR" %
%   B3:29/9  "TT-7119 LO TRIGGER BIT" %
% Rung: 477 %
SOR BST BST XIC B3:29/9 NXB XIC B9:28/10 XIO B3:0/1 BND OTE B9:28/10 NXB BST XIC B3:29/9 NXB XIC B9:28/11 XIO B3:0/1 XIO B3:0/0 BND OTE B9:28/11 BND EOR
%   B3:29/9  "TT-7119 LO TRIGGER BIT" %
%   B9:28/10  TT_7119_LO_ALM  "TT-7119 LO ALARM BIT" %
%   B3:0/1  ALARM_RESET  "ALARM RESET" %
%   B9:28/11  TT_7119_LO_ALT  "TT-7119 LO ALERT BIT" %
%   B3:0/0  ALARM_SILENCE  "ALARM SILENCE PUSHBUTTON" %
% Rung: 478 %
SOR GRT N11:115 0 GRT F8:57 F10:115 XIO B3:0/1 BST TON T4:115 1.0 0 0 NXB XIC T4:115/DN OSR B3:29/10 OTE B3:29/11 BND EOR
%   N11:115  TT_7119_HIALM_DLY_SP  "TT-7119 HI ALARM DELAY SP FROM HMI" %
%   F8:57  TT_7119_SCI  "TT-7119 SCALED INPUT" %
%   F10:115  TT_7119_HIALM_SP  "TT-7119 HI ALARM SP" %
%   B3:0/1  ALARM_RESET  "ALARM RESET" %
%   T4:115  TT_7119_HIALM_DLY_TM  "TT-7119 HI ALARM DELAY" %
%   B3:29/10  "OSR" %
%   B3:29/11  "TT-7119 HI TRIGGER BIT" %

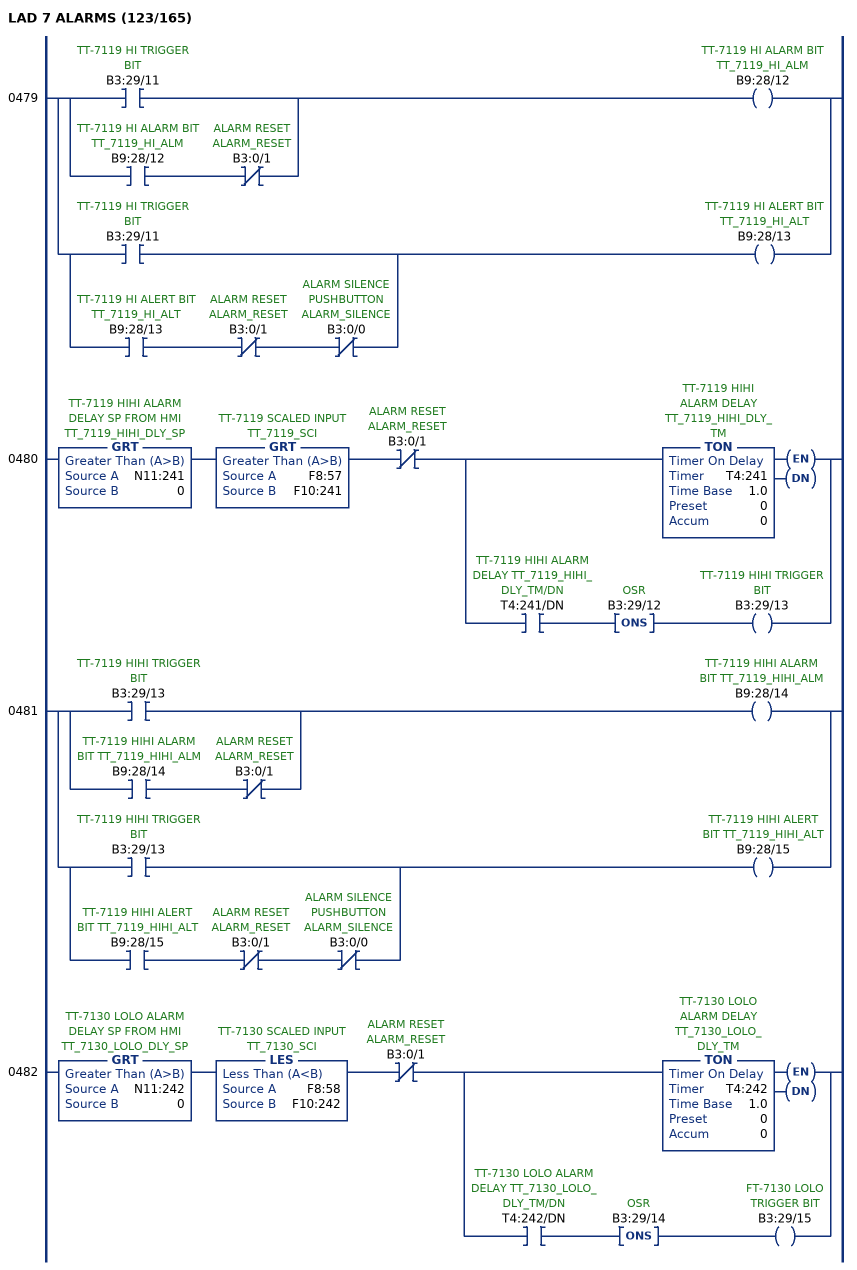
% Rung: 479 %
SOR BST BST XIC B3:29/11 NXB XIC B9:28/12 XIO B3:0/1 BND OTE B9:28/12 NXB BST XIC B3:29/11 NXB XIC B9:28/13 XIO B3:0/1 XIO B3:0/0 BND OTE B9:28/13 BND EOR
%   B3:29/11  "TT-7119 HI TRIGGER BIT" %
%   B9:28/12  TT_7119_HI_ALM  "TT-7119 HI ALARM BIT" %
%   B3:0/1  ALARM_RESET  "ALARM RESET" %
%   B9:28/13  TT_7119_HI_ALT  "TT-7119 HI ALERT BIT" %
%   B3:0/0  ALARM_SILENCE  "ALARM SILENCE PUSHBUTTON" %
% Rung: 480 %
SOR GRT N11:241 0 GRT F8:57 F10:241 XIO B3:0/1 BST TON T4:241 1.0 0 0 NXB XIC T4:241/DN OSR B3:29/12 OTE B3:29/13 BND EOR
%   N11:241  TT_7119_HIHI_DLY_SP  "TT-7119 HIHI ALARM DELAY SP FROM HMI" %
%   F8:57  TT_7119_SCI  "TT-7119 SCALED INPUT" %
%   F10:241  TT_7119_HIHI_SP  "TT-7119 HIHI ALARM SP" %
%   B3:0/1  ALARM_RESET  "ALARM RESET" %
%   T4:241  TT_7119_HIHI_DLY_TM  "TT-7119 HIHI ALARM DELAY" %
%   B3:29/12  "OSR" %
%   B3:29/13  "TT-7119 HIHI TRIGGER BIT" %
% Rung: 481 %
SOR BST BST XIC B3:29/13 NXB XIC B9:28/14 XIO B3:0/1 BND OTE B9:28/14 NXB BST XIC B3:29/13 NXB XIC B9:28/15 XIO B3:0/1 XIO B3:0/0 BND OTE B9:28/15 BND EOR
%   B3:29/13  "TT-7119 HIHI TRIGGER BIT" %
%   B9:28/14  TT_7119_HIHI_ALM  "TT-7119 HIHI ALARM BIT" %
%   B3:0/1  ALARM_RESET  "ALARM RESET" %
%   B9:28/15  TT_7119_HIHI_ALT  "TT-7119 HIHI ALERT BIT" %
%   B3:0/0  ALARM_SILENCE  "ALARM SILENCE PUSHBUTTON" %
% Rung: 482 %
SOR GRT N11:242 0 LES F8:58 F10:242 XIO B3:0/1 BST TON T4:242 1.0 0 0 NXB XIC T4:242/DN OSR B3:29/14 OTE B3:29/15 BND EOR
%   N11:242  TT_7130_LOLO_DLY_SP  "TT-7130 LOLO ALARM DELAY SP FROM HMI" %
%   F8:58  TT_7130_SCI  "TT-7130 SCALED INPUT" %
%   F10:242  TT_7130_LOLO_SP  "TT-7130 LOLO ALARM SP" %
%   B3:0/1  ALARM_RESET  "ALARM RESET" %
%   T4:242  TT_7130_LOLO_DLY_TM  "TT-7130 LOLO ALARM DELAY" %
%   B3:29/14  "OSR" %
%   B3:29/15  "FT-7130 LOLO TRIGGER BIT" %

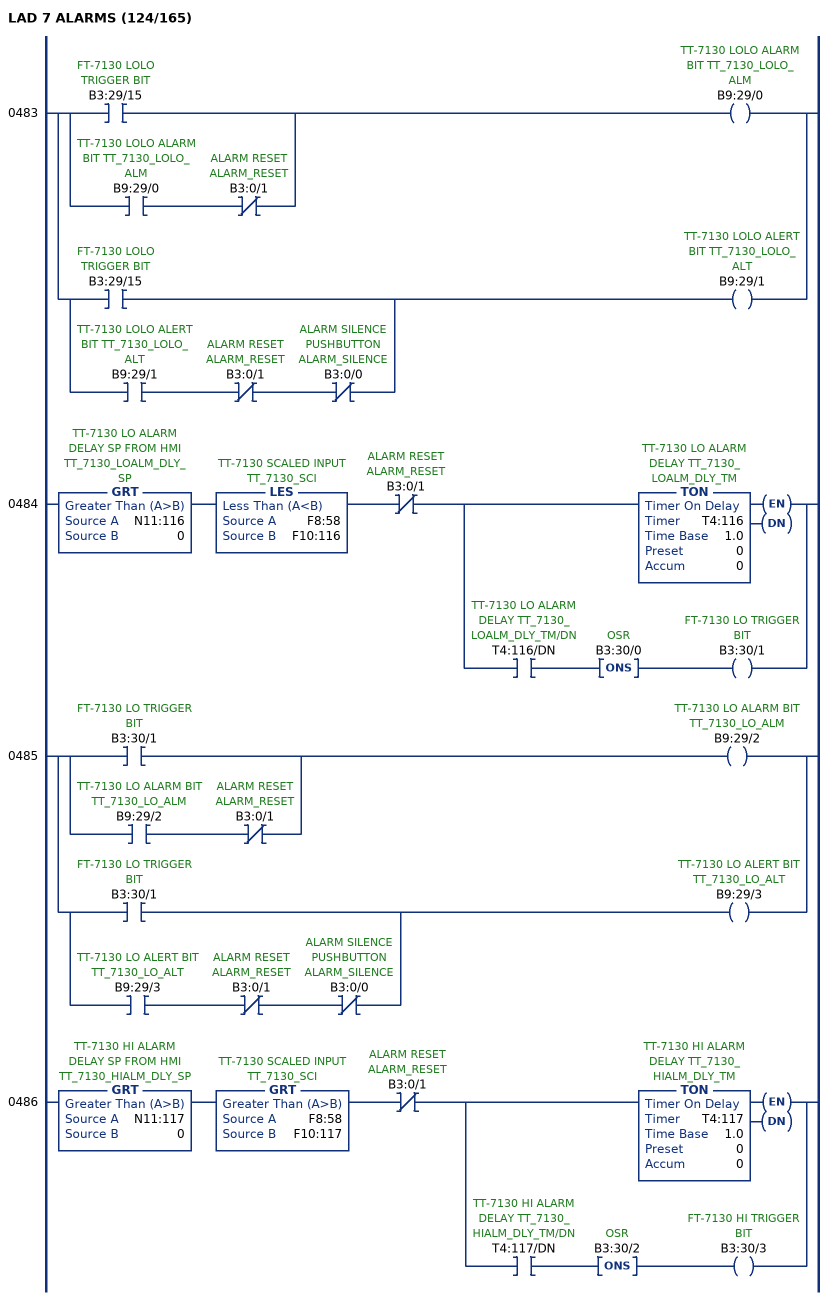
% Rung: 483 %
SOR BST BST XIC B3:29/15 NXB XIC B9:29/0 XIO B3:0/1 BND OTE B9:29/0 NXB BST XIC B3:29/15 NXB XIC B9:29/1 XIO B3:0/1 XIO B3:0/0 BND OTE B9:29/1 BND EOR
%   B3:29/15  "FT-7130 LOLO TRIGGER BIT" %
%   B9:29/0  TT_7130_LOLO_ALM  "TT-7130 LOLO ALARM BIT" %
%   B3:0/1  ALARM_RESET  "ALARM RESET" %
%   B9:29/1  TT_7130_LOLO_ALT  "TT-7130 LOLO ALERT BIT" %
%   B3:0/0  ALARM_SILENCE  "ALARM SILENCE PUSHBUTTON" %
% Rung: 484 %
SOR GRT N11:116 0 LES F8:58 F10:116 XIO B3:0/1 BST TON T4:116 1.0 0 0 NXB XIC T4:116/DN OSR B3:30/0 OTE B3:30/1 BND EOR
%   N11:116  TT_7130_LOALM_DLY_SP  "TT-7130 LO ALARM DELAY SP FROM HMI" %
%   F8:58  TT_7130_SCI  "TT-7130 SCALED INPUT" %
%   F10:116  TT_7130_LOALM_SP  "TT-7130 LO ALARM SP" %
%   B3:0/1  ALARM_RESET  "ALARM RESET" %
%   T4:116  TT_7130_LOALM_DLY_TM  "TT-7130 LO ALARM DELAY" %
%   B3:30/0  "OSR" %
%   B3:30/1  "FT-7130 LO TRIGGER BIT" %
% Rung: 485 %
SOR BST BST XIC B3:30/1 NXB XIC B9:29/2 XIO B3:0/1 BND OTE B9:29/2 NXB BST XIC B3:30/1 NXB XIC B9:29/3 XIO B3:0/1 XIO B3:0/0 BND OTE B9:29/3 BND EOR
%   B3:30/1  "FT-7130 LO TRIGGER BIT" %
%   B9:29/2  TT_7130_LO_ALM  "TT-7130 LO ALARM BIT" %
%   B3:0/1  ALARM_RESET  "ALARM RESET" %
%   B9:29/3  TT_7130_LO_ALT  "TT-7130 LO ALERT BIT" %
%   B3:0/0  ALARM_SILENCE  "ALARM SILENCE PUSHBUTTON" %
% Rung: 486 %
SOR GRT N11:117 0 GRT F8:58 F10:117 XIO B3:0/1 BST TON T4:117 1.0 0 0 NXB XIC T4:117/DN OSR B3:30/2 OTE B3:30/3 BND EOR
%   N11:117  TT_7130_HIALM_DLY_SP  "TT-7130 HI ALARM DELAY SP FROM HMI" %
%   F8:58  TT_7130_SCI  "TT-7130 SCALED INPUT" %
%   F10:117  TT_7130_HIALM_SP  "TT-7130 HI ALARM SP" %
%   B3:0/1  ALARM_RESET  "ALARM RESET" %
%   T4:117  TT_7130_HIALM_DLY_TM  "TT-7130 HI ALARM DELAY" %
%   B3:30/2  "OSR" %
%   B3:30/3  "FT-7130 HI TRIGGER BIT" %

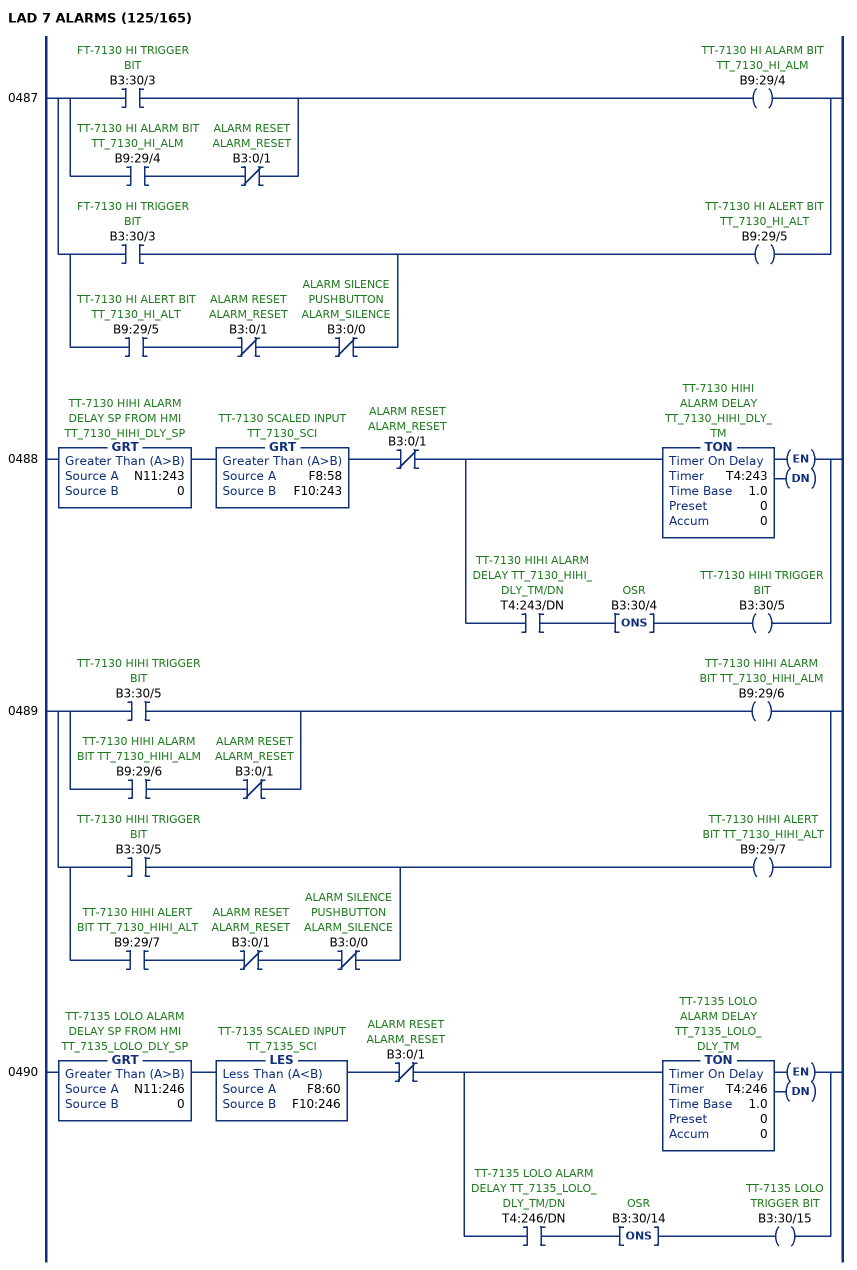
% Rung: 487 %
SOR BST BST XIC B3:30/3 NXB XIC B9:29/4 XIO B3:0/1 BND OTE B9:29/4 NXB BST XIC B3:30/3 NXB XIC B9:29/5 XIO B3:0/1 XIO B3:0/0 BND OTE B9:29/5 BND EOR
%   B3:30/3  "FT-7130 HI TRIGGER BIT" %
%   B9:29/4  TT_7130_HI_ALM  "TT-7130 HI ALARM BIT" %
%   B3:0/1  ALARM_RESET  "ALARM RESET" %
%   B9:29/5  TT_7130_HI_ALT  "TT-7130 HI ALERT BIT" %
%   B3:0/0  ALARM_SILENCE  "ALARM SILENCE PUSHBUTTON" %
% Rung: 488 %
SOR GRT N11:243 0 GRT F8:58 F10:243 XIO B3:0/1 BST TON T4:243 1.0 0 0 NXB XIC T4:243/DN OSR B3:30/4 OTE B3:30/5 BND EOR
%   N11:243  TT_7130_HIHI_DLY_SP  "TT-7130 HIHI ALARM DELAY SP FROM HMI" %
%   F8:58  TT_7130_SCI  "TT-7130 SCALED INPUT" %
%   F10:243  TT_7130_HIHI_SP  "TT-7130 HIHI ALARM SP" %
%   B3:0/1  ALARM_RESET  "ALARM RESET" %
%   T4:243  TT_7130_HIHI_DLY_TM  "TT-7130 HIHI ALARM DELAY" %
%   B3:30/4  "OSR" %
%   B3:30/5  "TT-7130 HIHI TRIGGER BIT" %
% Rung: 489 %
SOR BST BST XIC B3:30/5 NXB XIC B9:29/6 XIO B3:0/1 BND OTE B9:29/6 NXB BST XIC B3:30/5 NXB XIC B9:29/7 XIO B3:0/1 XIO B3:0/0 BND OTE B9:29/7 BND EOR
%   B3:30/5  "TT-7130 HIHI TRIGGER BIT" %
%   B9:29/6  TT_7130_HIHI_ALM  "TT-7130 HIHI ALARM BIT" %
%   B3:0/1  ALARM_RESET  "ALARM RESET" %
%   B9:29/7  TT_7130_HIHI_ALT  "TT-7130 HIHI ALERT BIT" %
%   B3:0/0  ALARM_SILENCE  "ALARM SILENCE PUSHBUTTON" %
% Rung: 490 %
SOR GRT N11:246 0 LES F8:60 F10:246 XIO B3:0/1 BST TON T4:246 1.0 0 0 NXB XIC T4:246/DN OSR B3:30/14 OTE B3:30/15 BND EOR
%   N11:246  TT_7135_LOLO_DLY_SP  "TT-7135 LOLO ALARM DELAY SP FROM HMI" %
%   F8:60  TT_7135_SCI  "TT-7135 SCALED INPUT" %
%   F10:246  TT_7135_LOLO_SP  "TT-7135 LOLO ALARM SP" %
%   B3:0/1  ALARM_RESET  "ALARM RESET" %
%   T4:246  TT_7135_LOLO_DLY_TM  "TT-7135 LOLO ALARM DELAY" %
%   B3:30/14  "OSR" %
%   B3:30/15  "TT-7135 LOLO TRIGGER BIT" %

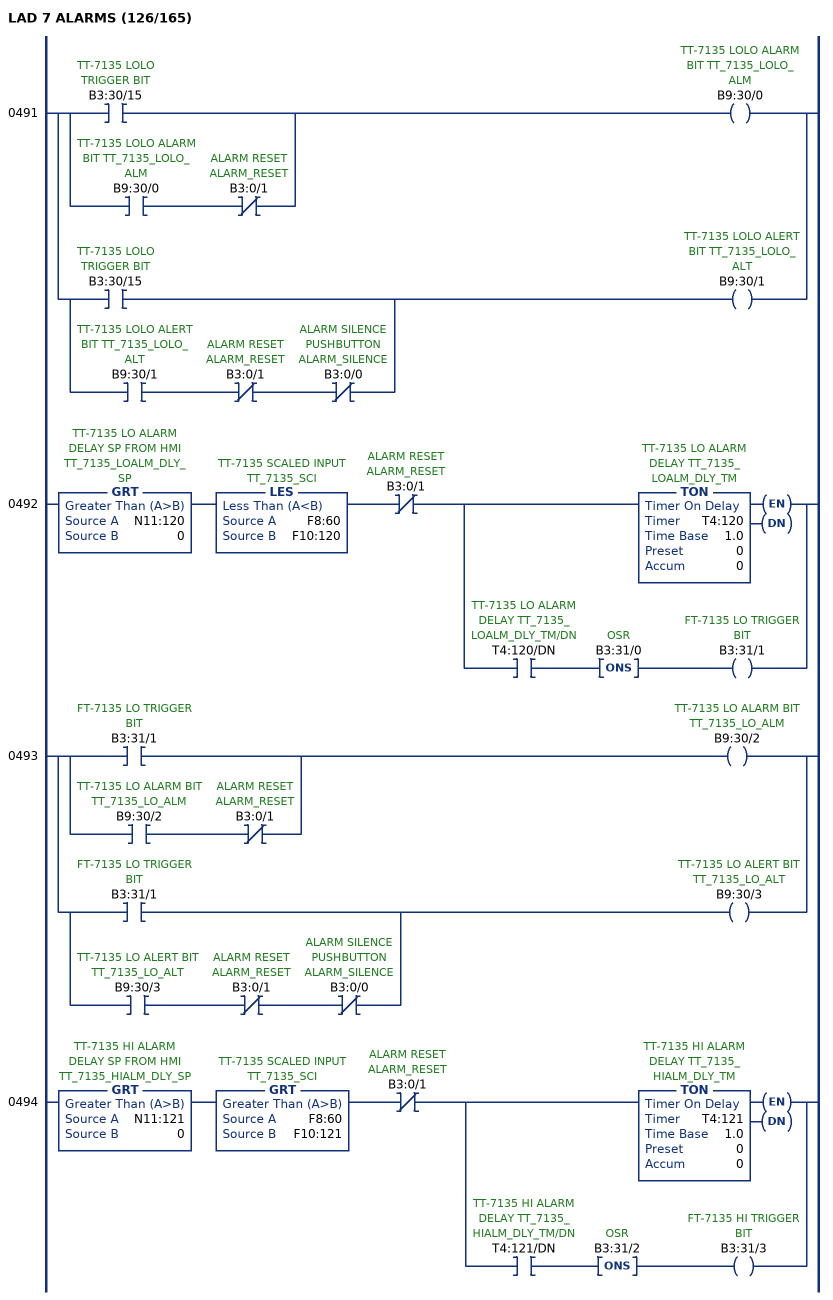
% Rung: 491 %
SOR BST BST XIC B3:30/15 NXB XIC B9:30/0 XIO B3:0/1 BND OTE B9:30/0 NXB BST XIC B3:30/15 NXB XIC B9:30/1 XIO B3:0/1 XIO B3:0/0 BND OTE B9:30/1 BND EOR
%   B3:30/15  "TT-7135 LOLO TRIGGER BIT" %
%   B9:30/0  TT_7135_LOLO_ALM  "TT-7135 LOLO ALARM BIT" %
%   B3:0/1  ALARM_RESET  "ALARM RESET" %
%   B9:30/1  TT_7135_LOLO_ALT  "TT-7135 LOLO ALERT BIT" %
%   B3:0/0  ALARM_SILENCE  "ALARM SILENCE PUSHBUTTON" %
% Rung: 492 %
SOR GRT N11:120 0 LES F8:60 F10:120 XIO B3:0/1 BST TON T4:120 1.0 0 0 NXB XIC T4:120/DN OSR B3:31/0 OTE B3:31/1 BND EOR
%   N11:120  TT_7135_LOALM_DLY_SP  "TT-7135 LO ALARM DELAY SP FROM HMI" %
%   F8:60  TT_7135_SCI  "TT-7135 SCALED INPUT" %
%   F10:120  TT_7135_LOALM_SP  "TT-7135 LO ALARM SP" %
%   B3:0/1  ALARM_RESET  "ALARM RESET" %
%   T4:120  TT_7135_LOALM_DLY_TM  "TT-7135 LO ALARM DELAY" %
%   B3:31/0  "OSR" %
%   B3:31/1  "FT-7135 LO TRIGGER BIT" %
% Rung: 493 %
SOR BST BST XIC B3:31/1 NXB XIC B9:30/2 XIO B3:0/1 BND OTE B9:30/2 NXB BST XIC B3:31/1 NXB XIC B9:30/3 XIO B3:0/1 XIO B3:0/0 BND OTE B9:30/3 BND EOR
%   B3:31/1  "FT-7135 LO TRIGGER BIT" %
%   B9:30/2  TT_7135_LO_ALM  "TT-7135 LO ALARM BIT" %
%   B3:0/1  ALARM_RESET  "ALARM RESET" %
%   B9:30/3  TT_7135_LO_ALT  "TT-7135 LO ALERT BIT" %
%   B3:0/0  ALARM_SILENCE  "ALARM SILENCE PUSHBUTTON" %
% Rung: 494 %
SOR GRT N11:121 0 GRT F8:60 F10:121 XIO B3:0/1 BST TON T4:121 1.0 0 0 NXB XIC T4:121/DN OSR B3:31/2 OTE B3:31/3 BND EOR
%   N11:121  TT_7135_HIALM_DLY_SP  "TT-7135 HI ALARM DELAY SP FROM HMI" %
%   F8:60  TT_7135_SCI  "TT-7135 SCALED INPUT" %
%   F10:121  TT_7135_HIALM_SP  "TT-7135 HI ALARM SP" %
%   B3:0/1  ALARM_RESET  "ALARM RESET" %
%   T4:121  TT_7135_HIALM_DLY_TM  "TT-7135 HI ALARM DELAY" %
%   B3:31/2  "OSR" %
%   B3:31/3  "FT-7135 HI TRIGGER BIT" %

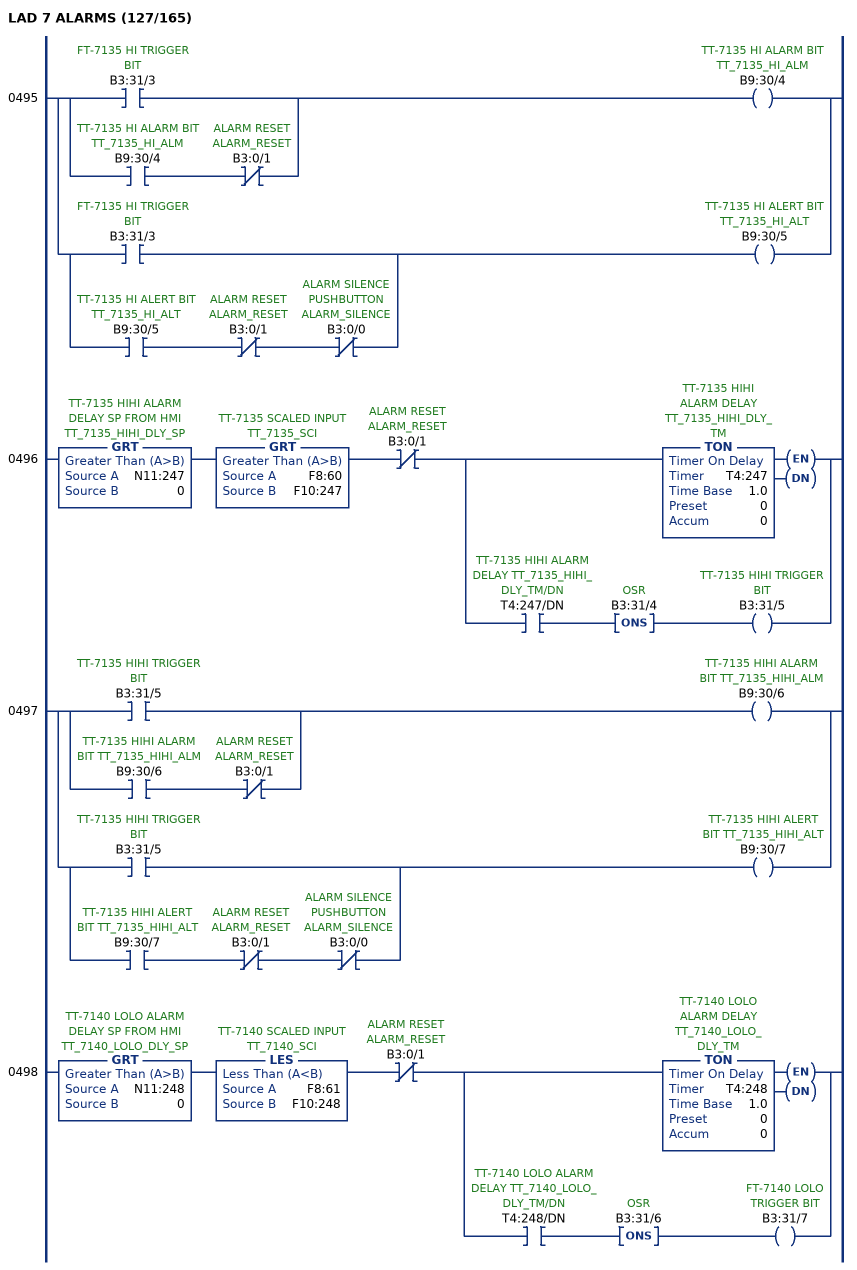
% Rung: 495 %
SOR BST BST XIC B3:31/3 NXB XIC B9:30/4 XIO B3:0/1 BND OTE B9:30/4 NXB BST XIC B3:31/3 NXB XIC B9:30/5 XIO B3:0/1 XIO B3:0/0 BND OTE B9:30/5 BND EOR
%   B3:31/3  "FT-7135 HI TRIGGER BIT" %
%   B9:30/4  TT_7135_HI_ALM  "TT-7135 HI ALARM BIT" %
%   B3:0/1  ALARM_RESET  "ALARM RESET" %
%   B9:30/5  TT_7135_HI_ALT  "TT-7135 HI ALERT BIT" %
%   B3:0/0  ALARM_SILENCE  "ALARM SILENCE PUSHBUTTON" %
% Rung: 496 %
SOR GRT N11:247 0 GRT F8:60 F10:247 XIO B3:0/1 BST TON T4:247 1.0 0 0 NXB XIC T4:247/DN OSR B3:31/4 OTE B3:31/5 BND EOR
%   N11:247  TT_7135_HIHI_DLY_SP  "TT-7135 HIHI ALARM DELAY SP FROM HMI" %
%   F8:60  TT_7135_SCI  "TT-7135 SCALED INPUT" %
%   F10:247  TT_7135_HIHI_SP  "TT-7135 HIHI ALARM SP" %
%   B3:0/1  ALARM_RESET  "ALARM RESET" %
%   T4:247  TT_7135_HIHI_DLY_TM  "TT-7135 HIHI ALARM DELAY" %
%   B3:31/4  "OSR" %
%   B3:31/5  "TT-7135 HIHI TRIGGER BIT" %
% Rung: 497 %
SOR BST BST XIC B3:31/5 NXB XIC B9:30/6 XIO B3:0/1 BND OTE B9:30/6 NXB BST XIC B3:31/5 NXB XIC B9:30/7 XIO B3:0/1 XIO B3:0/0 BND OTE B9:30/7 BND EOR
%   B3:31/5  "TT-7135 HIHI TRIGGER BIT" %
%   B9:30/6  TT_7135_HIHI_ALM  "TT-7135 HIHI ALARM BIT" %
%   B3:0/1  ALARM_RESET  "ALARM RESET" %
%   B9:30/7  TT_7135_HIHI_ALT  "TT-7135 HIHI ALERT BIT" %
%   B3:0/0  ALARM_SILENCE  "ALARM SILENCE PUSHBUTTON" %
% Rung: 498 %
SOR GRT N11:248 0 LES F8:61 F10:248 XIO B3:0/1 BST TON T4:248 1.0 0 0 NXB XIC T4:248/DN OSR B3:31/6 OTE B3:31/7 BND EOR
%   N11:248  TT_7140_LOLO_DLY_SP  "TT-7140 LOLO ALARM DELAY SP FROM HMI" %
%   F8:61  TT_7140_SCI  "TT-7140 SCALED INPUT" %
%   F10:248  TT_7140_LOLO_SP  "TT-7140 LOLO ALARM SP" %
%   B3:0/1  ALARM_RESET  "ALARM RESET" %
%   T4:248  TT_7140_LOLO_DLY_TM  "TT-7140 LOLO ALARM DELAY" %
%   B3:31/6  "OSR" %
%   B3:31/7  "FT-7140 LOLO TRIGGER BIT" %

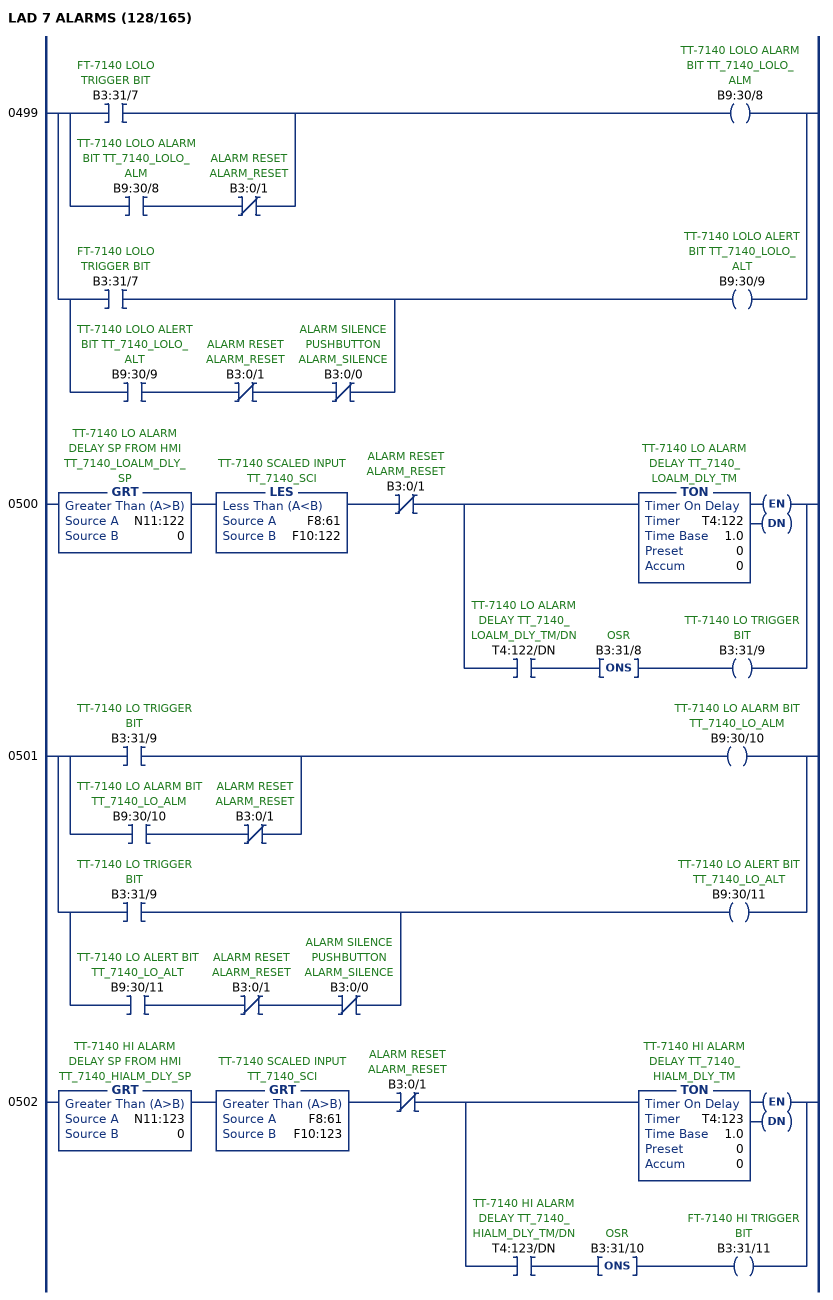
% Rung: 499 %
SOR BST BST XIC B3:31/7 NXB XIC B9:30/8 XIO B3:0/1 BND OTE B9:30/8 NXB BST XIC B3:31/7 NXB XIC B9:30/9 XIO B3:0/1 XIO B3:0/0 BND OTE B9:30/9 BND EOR
%   B3:31/7  "FT-7140 LOLO TRIGGER BIT" %
%   B9:30/8  TT_7140_LOLO_ALM  "TT-7140 LOLO ALARM BIT" %
%   B3:0/1  ALARM_RESET  "ALARM RESET" %
%   B9:30/9  TT_7140_LOLO_ALT  "TT-7140 LOLO ALERT BIT" %
%   B3:0/0  ALARM_SILENCE  "ALARM SILENCE PUSHBUTTON" %
% Rung: 500 %
SOR GRT N11:122 0 LES F8:61 F10:122 XIO B3:0/1 BST TON T4:122 1.0 0 0 NXB XIC T4:122/DN OSR B3:31/8 OTE B3:31/9 BND EOR
%   N11:122  TT_7140_LOALM_DLY_SP  "TT-7140 LO ALARM DELAY SP FROM HMI" %
%   F8:61  TT_7140_SCI  "TT-7140 SCALED INPUT" %
%   F10:122  TT_7140_LOALM_SP  "TT-7140 LO ALARM SP" %
%   B3:0/1  ALARM_RESET  "ALARM RESET" %
%   T4:122  TT_7140_LOALM_DLY_TM  "TT-7140 LO ALARM DELAY" %
%   B3:31/8  "OSR" %
%   B3:31/9  "TT-7140 LO TRIGGER BIT" %
% Rung: 501 %
SOR BST BST XIC B3:31/9 NXB XIC B9:30/10 XIO B3:0/1 BND OTE B9:30/10 NXB BST XIC B3:31/9 NXB XIC B9:30/11 XIO B3:0/1 XIO B3:0/0 BND OTE B9:30/11 BND EOR
%   B3:31/9  "TT-7140 LO TRIGGER BIT" %
%   B9:30/10  TT_7140_LO_ALM  "TT-7140 LO ALARM BIT" %
%   B3:0/1  ALARM_RESET  "ALARM RESET" %
%   B9:30/11  TT_7140_LO_ALT  "TT-7140 LO ALERT BIT" %
%   B3:0/0  ALARM_SILENCE  "ALARM SILENCE PUSHBUTTON" %
% Rung: 502 %
SOR GRT N11:123 0 GRT F8:61 F10:123 XIO B3:0/1 BST TON T4:123 1.0 0 0 NXB XIC T4:123/DN OSR B3:31/10 OTE B3:31/11 BND EOR
%   N11:123  TT_7140_HIALM_DLY_SP  "TT-7140 HI ALARM DELAY SP FROM HMI" %
%   F8:61  TT_7140_SCI  "TT-7140 SCALED INPUT" %
%   F10:123  TT_7140_HIALM_SP  "TT-7140 HI ALARM SP" %
%   B3:0/1  ALARM_RESET  "ALARM RESET" %
%   T4:123  TT_7140_HIALM_DLY_TM  "TT-7140 HI ALARM DELAY" %
%   B3:31/10  "OSR" %
%   B3:31/11  "FT-7140 HI TRIGGER BIT" %

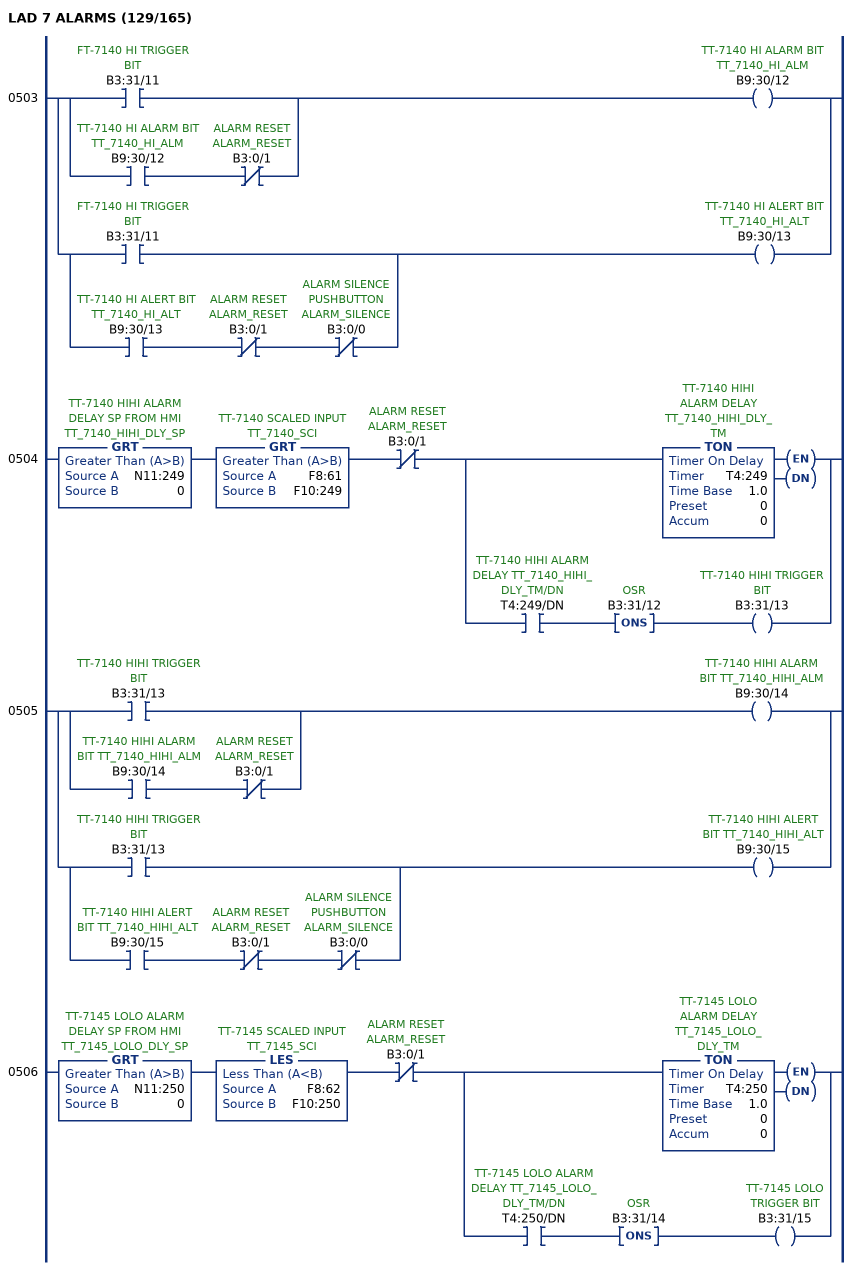
% Rung: 503 %
SOR BST BST XIC B3:31/11 NXB XIC B9:30/12 XIO B3:0/1 BND OTE B9:30/12 NXB BST XIC B3:31/11 NXB XIC B9:30/13 XIO B3:0/1 XIO B3:0/0 BND OTE B9:30/13 BND EOR
%   B3:31/11  "FT-7140 HI TRIGGER BIT" %
%   B9:30/12  TT_7140_HI_ALM  "TT-7140 HI ALARM BIT" %
%   B3:0/1  ALARM_RESET  "ALARM RESET" %
%   B9:30/13  TT_7140_HI_ALT  "TT-7140 HI ALERT BIT" %
%   B3:0/0  ALARM_SILENCE  "ALARM SILENCE PUSHBUTTON" %
% Rung: 504 %
SOR GRT N11:249 0 GRT F8:61 F10:249 XIO B3:0/1 BST TON T4:249 1.0 0 0 NXB XIC T4:249/DN OSR B3:31/12 OTE B3:31/13 BND EOR
%   N11:249  TT_7140_HIHI_DLY_SP  "TT-7140 HIHI ALARM DELAY SP FROM HMI" %
%   F8:61  TT_7140_SCI  "TT-7140 SCALED INPUT" %
%   F10:249  TT_7140_HIHI_SP  "TT-7140 HIHI ALARM SP" %
%   B3:0/1  ALARM_RESET  "ALARM RESET" %
%   T4:249  TT_7140_HIHI_DLY_TM  "TT-7140 HIHI ALARM DELAY" %
%   B3:31/12  "OSR" %
%   B3:31/13  "TT-7140 HIHI TRIGGER BIT" %
% Rung: 505 %
SOR BST BST XIC B3:31/13 NXB XIC B9:30/14 XIO B3:0/1 BND OTE B9:30/14 NXB BST XIC B3:31/13 NXB XIC B9:30/15 XIO B3:0/1 XIO B3:0/0 BND OTE B9:30/15 BND EOR
%   B3:31/13  "TT-7140 HIHI TRIGGER BIT" %
%   B9:30/14  TT_7140_HIHI_ALM  "TT-7140 HIHI ALARM BIT" %
%   B3:0/1  ALARM_RESET  "ALARM RESET" %
%   B9:30/15  TT_7140_HIHI_ALT  "TT-7140 HIHI ALERT BIT" %
%   B3:0/0  ALARM_SILENCE  "ALARM SILENCE PUSHBUTTON" %
% Rung: 506 %
SOR GRT N11:250 0 LES F8:62 F10:250 XIO B3:0/1 BST TON T4:250 1.0 0 0 NXB XIC T4:250/DN OSR B3:31/14 OTE B3:31/15 BND EOR
%   N11:250  TT_7145_LOLO_DLY_SP  "TT-7145 LOLO ALARM DELAY SP FROM HMI" %
%   F8:62  TT_7145_SCI  "TT-7145 SCALED INPUT" %
%   F10:250  TT_7145_LOLO_SP  "TT-7145 LOLO ALARM SP" %
%   B3:0/1  ALARM_RESET  "ALARM RESET" %
%   T4:250  TT_7145_LOLO_DLY_TM  "TT-7145 LOLO ALARM DELAY" %
%   B3:31/14  "OSR" %
%   B3:31/15  "TT-7145 LOLO TRIGGER BIT" %

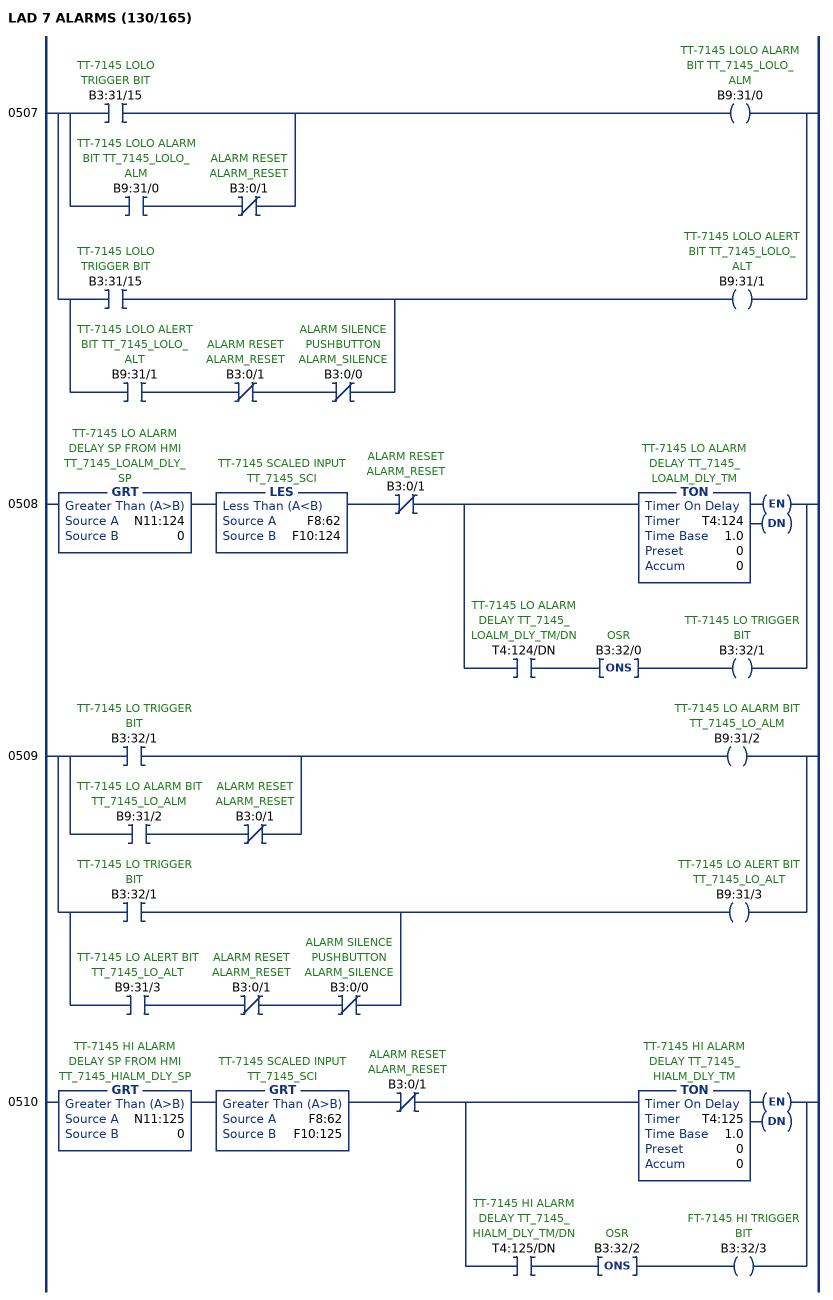
% Rung: 507 %
SOR BST BST XIC B3:31/15 NXB XIC B9:31/0 XIO B3:0/1 BND OTE B9:31/0 NXB BST XIC B3:31/15 NXB XIC B9:31/1 XIO B3:0/1 XIO B3:0/0 BND OTE B9:31/1 BND EOR
%   B3:31/15  "TT-7145 LOLO TRIGGER BIT" %
%   B9:31/0  TT_7145_LOLO_ALM  "TT-7145 LOLO ALARM BIT" %
%   B3:0/1  ALARM_RESET  "ALARM RESET" %
%   B9:31/1  TT_7145_LOLO_ALT  "TT-7145 LOLO ALERT BIT" %
%   B3:0/0  ALARM_SILENCE  "ALARM SILENCE PUSHBUTTON" %
% Rung: 508 %
SOR GRT N11:124 0 LES F8:62 F10:124 XIO B3:0/1 BST TON T4:124 1.0 0 0 NXB XIC T4:124/DN OSR B3:32/0 OTE B3:32/1 BND EOR
%   N11:124  TT_7145_LOALM_DLY_SP  "TT-7145 LO ALARM DELAY SP FROM HMI" %
%   F8:62  TT_7145_SCI  "TT-7145 SCALED INPUT" %
%   F10:124  TT_7145_LOALM_SP  "TT-7145 LO ALARM SP" %
%   B3:0/1  ALARM_RESET  "ALARM RESET" %
%   T4:124  TT_7145_LOALM_DLY_TM  "TT-7145 LO ALARM DELAY" %
%   B3:32/0  "OSR" %
%   B3:32/1  "TT-7145 LO TRIGGER BIT" %
% Rung: 509 %
SOR BST BST XIC B3:32/1 NXB XIC B9:31/2 XIO B3:0/1 BND OTE B9:31/2 NXB BST XIC B3:32/1 NXB XIC B9:31/3 XIO B3:0/1 XIO B3:0/0 BND OTE B9:31/3 BND EOR
%   B3:32/1  "TT-7145 LO TRIGGER BIT" %
%   B9:31/2  TT_7145_LO_ALM  "TT-7145 LO ALARM BIT" %
%   B3:0/1  ALARM_RESET  "ALARM RESET" %
%   B9:31/3  TT_7145_LO_ALT  "TT-7145 LO ALERT BIT" %
%   B3:0/0  ALARM_SILENCE  "ALARM SILENCE PUSHBUTTON" %
% Rung: 510 %
SOR GRT N11:125 0 GRT F8:62 F10:125 XIO B3:0/1 BST TON T4:125 1.0 0 0 NXB XIC T4:125/DN OSR B3:32/2 OTE B3:32/3 BND EOR
%   N11:125  TT_7145_HIALM_DLY_SP  "TT-7145 HI ALARM DELAY SP FROM HMI" %
%   F8:62  TT_7145_SCI  "TT-7145 SCALED INPUT" %
%   F10:125  TT_7145_HIALM_SP  "TT-7145 HI ALARM SP" %
%   B3:0/1  ALARM_RESET  "ALARM RESET" %
%   T4:125  TT_7145_HIALM_DLY_TM  "TT-7145 HI ALARM DELAY" %
%   B3:32/2  "OSR" %
%   B3:32/3  "FT-7145 HI TRIGGER BIT" %

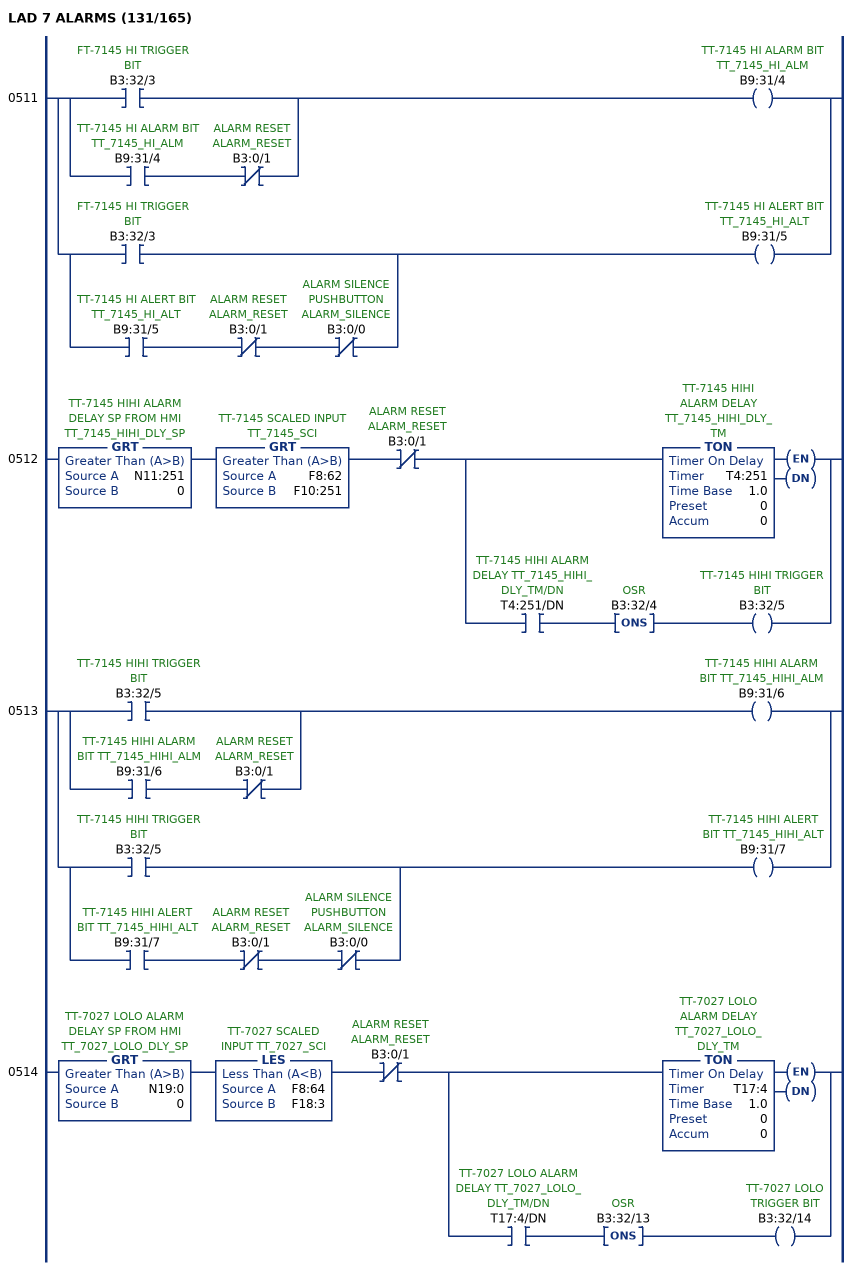
% Rung: 511 %
SOR BST BST XIC B3:32/3 NXB XIC B9:31/4 XIO B3:0/1 BND OTE B9:31/4 NXB BST XIC B3:32/3 NXB XIC B9:31/5 XIO B3:0/1 XIO B3:0/0 BND OTE B9:31/5 BND EOR
%   B3:32/3  "FT-7145 HI TRIGGER BIT" %
%   B9:31/4  TT_7145_HI_ALM  "TT-7145 HI ALARM BIT" %
%   B3:0/1  ALARM_RESET  "ALARM RESET" %
%   B9:31/5  TT_7145_HI_ALT  "TT-7145 HI ALERT BIT" %
%   B3:0/0  ALARM_SILENCE  "ALARM SILENCE PUSHBUTTON" %
% Rung: 512 %
SOR GRT N11:251 0 GRT F8:62 F10:251 XIO B3:0/1 BST TON T4:251 1.0 0 0 NXB XIC T4:251/DN OSR B3:32/4 OTE B3:32/5 BND EOR
%   N11:251  TT_7145_HIHI_DLY_SP  "TT-7145 HIHI ALARM DELAY SP FROM HMI" %
%   F8:62  TT_7145_SCI  "TT-7145 SCALED INPUT" %
%   F10:251  TT_7145_HIHI_SP  "TT-7145 HIHI ALARM SP" %
%   B3:0/1  ALARM_RESET  "ALARM RESET" %
%   T4:251  TT_7145_HIHI_DLY_TM  "TT-7145 HIHI ALARM DELAY" %
%   B3:32/4  "OSR" %
%   B3:32/5  "TT-7145 HIHI TRIGGER BIT" %
% Rung: 513 %
SOR BST BST XIC B3:32/5 NXB XIC B9:31/6 XIO B3:0/1 BND OTE B9:31/6 NXB BST XIC B3:32/5 NXB XIC B9:31/7 XIO B3:0/1 XIO B3:0/0 BND OTE B9:31/7 BND EOR
%   B3:32/5  "TT-7145 HIHI TRIGGER BIT" %
%   B9:31/6  TT_7145_HIHI_ALM  "TT-7145 HIHI ALARM BIT" %
%   B3:0/1  ALARM_RESET  "ALARM RESET" %
%   B9:31/7  TT_7145_HIHI_ALT  "TT-7145 HIHI ALERT BIT" %
%   B3:0/0  ALARM_SILENCE  "ALARM SILENCE PUSHBUTTON" %
% Rung: 514 %
SOR GRT N19:0 0 LES F8:64 F18:3 XIO B3:0/1 BST TON T17:4 1.0 0 0 NXB XIC T17:4/DN OSR B3:32/13 OTE B3:32/14 BND EOR
%   N19:0  TT_7027_LOLO_DLY_SP  "TT-7027 LOLO ALARM DELAY SP FROM HMI" %
%   F8:64  TT_7027_SCI  "TT-7027 SCALED INPUT" %
%   F18:3  TT_7027_LOLO_SP  "TT-7027 LOLO ALARM SP" %
%   B3:0/1  ALARM_RESET  "ALARM RESET" %
%   T17:4  TT_7027_LOLO_DLY_TM  "TT-7027 LOLO ALARM DELAY" %
%   B3:32/13  "OSR" %
%   B3:32/14  "TT-7027 LOLO TRIGGER BIT" %

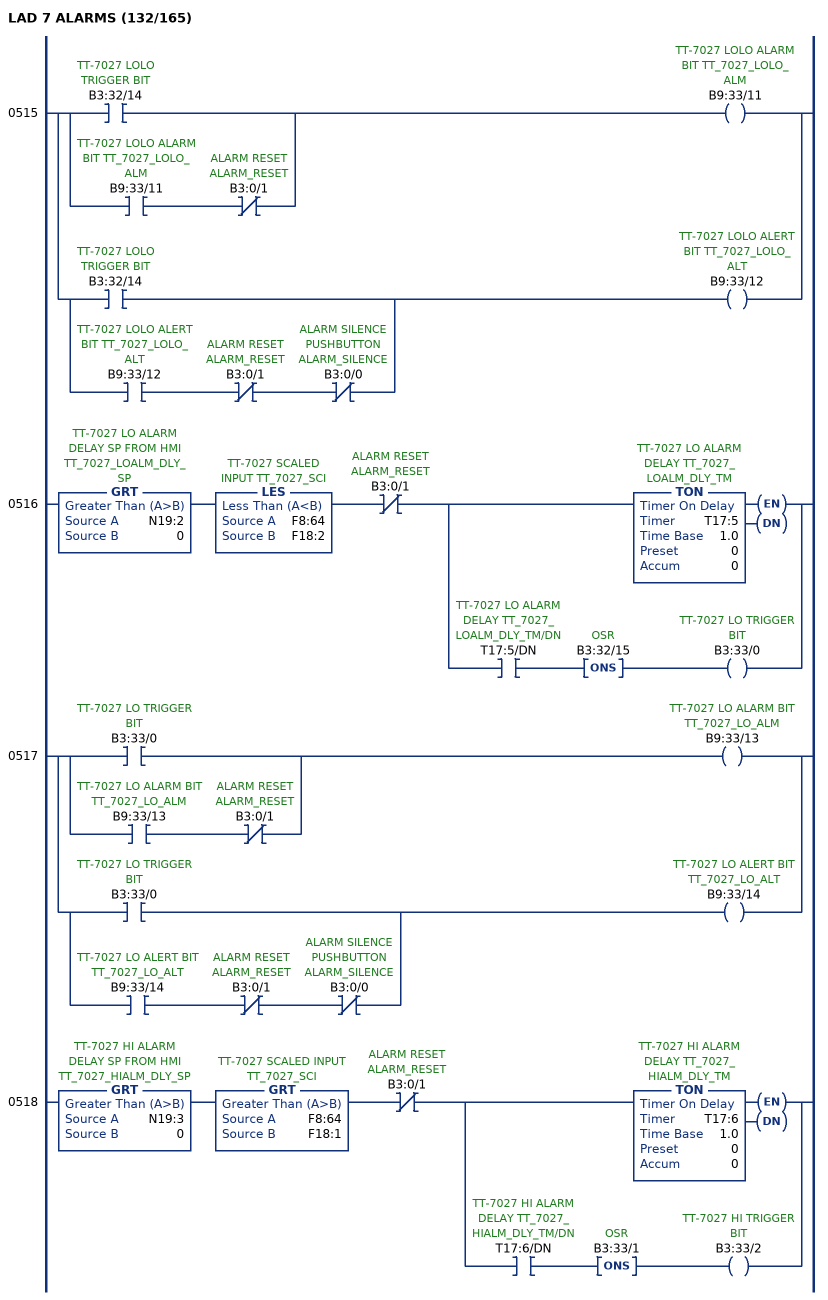
% Rung: 515 %
SOR BST BST XIC B3:32/14 NXB XIC B9:33/11 XIO B3:0/1 BND OTE B9:33/11 NXB BST XIC B3:32/14 NXB XIC B9:33/12 XIO B3:0/1 XIO B3:0/0 BND OTE B9:33/12 BND EOR
%   B3:32/14  "TT-7027 LOLO TRIGGER BIT" %
%   B9:33/11  TT_7027_LOLO_ALM  "TT-7027 LOLO ALARM BIT" %
%   B3:0/1  ALARM_RESET  "ALARM RESET" %
%   B9:33/12  TT_7027_LOLO_ALT  "TT-7027 LOLO ALERT BIT" %
%   B3:0/0  ALARM_SILENCE  "ALARM SILENCE PUSHBUTTON" %
% Rung: 516 %
SOR GRT N19:2 0 LES F8:64 F18:2 XIO B3:0/1 BST TON T17:5 1.0 0 0 NXB XIC T17:5/DN OSR B3:32/15 OTE B3:33/0 BND EOR
%   N19:2  TT_7027_LOALM_DLY_SP  "TT-7027 LO ALARM DELAY SP FROM HMI" %
%   F8:64  TT_7027_SCI  "TT-7027 SCALED INPUT" %
%   F18:2  TT_7027_LOALM_SP  "TT-7027 LO ALARM SP" %
%   B3:0/1  ALARM_RESET  "ALARM RESET" %
%   T17:5  TT_7027_LOALM_DLY_TM  "TT-7027 LO ALARM DELAY" %
%   B3:32/15  "OSR" %
%   B3:33/0  "TT-7027 LO TRIGGER BIT" %
% Rung: 517 %
SOR BST BST XIC B3:33/0 NXB XIC B9:33/13 XIO B3:0/1 BND OTE B9:33/13 NXB BST XIC B3:33/0 NXB XIC B9:33/14 XIO B3:0/1 XIO B3:0/0 BND OTE B9:33/14 BND EOR
%   B3:33/0  "TT-7027 LO TRIGGER BIT" %
%   B9:33/13  TT_7027_LO_ALM  "TT-7027 LO ALARM BIT" %
%   B3:0/1  ALARM_RESET  "ALARM RESET" %
%   B9:33/14  TT_7027_LO_ALT  "TT-7027 LO ALERT BIT" %
%   B3:0/0  ALARM_SILENCE  "ALARM SILENCE PUSHBUTTON" %
% Rung: 518 %
SOR GRT N19:3 0 GRT F8:64 F18:1 XIO B3:0/1 BST TON T17:6 1.0 0 0 NXB XIC T17:6/DN OSR B3:33/1 OTE B3:33/2 BND EOR
%   N19:3  TT_7027_HIALM_DLY_SP  "TT-7027 HI ALARM DELAY SP FROM HMI" %
%   F8:64  TT_7027_SCI  "TT-7027 SCALED INPUT" %
%   F18:1  TT_7027_HIALM_SP  "TT-7027 HI ALARM SP" %
%   B3:0/1  ALARM_RESET  "ALARM RESET" %
%   T17:6  TT_7027_HIALM_DLY_TM  "TT-7027 HI ALARM DELAY" %
%   B3:33/1  "OSR" %
%   B3:33/2  "TT-7027 HI TRIGGER BIT" %

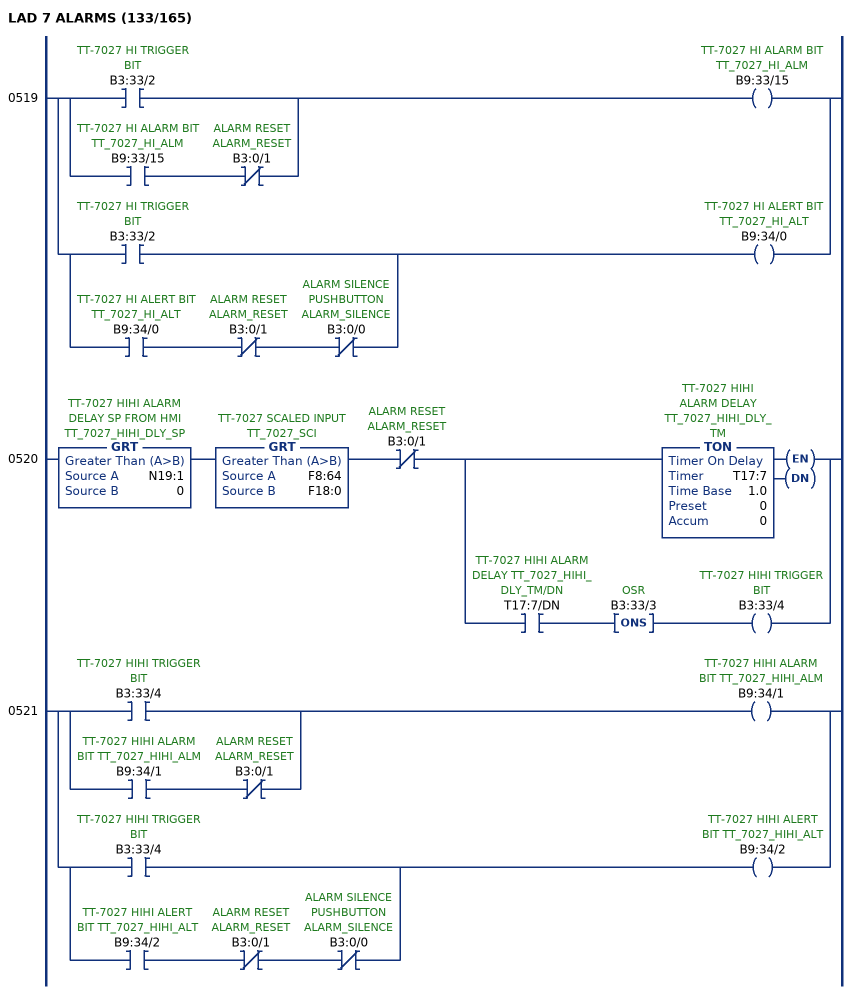
% Rung: 519 %
SOR BST BST XIC B3:33/2 NXB XIC B9:33/15 XIO B3:0/1 BND OTE B9:33/15 NXB BST XIC B3:33/2 NXB XIC B9:34/0 XIO B3:0/1 XIO B3:0/0 BND OTE B9:34/0 BND EOR
%   B3:33/2  "TT-7027 HI TRIGGER BIT" %
%   B9:33/15  TT_7027_HI_ALM  "TT-7027 HI ALARM BIT" %
%   B3:0/1  ALARM_RESET  "ALARM RESET" %
%   B9:34/0  TT_7027_HI_ALT  "TT-7027 HI ALERT BIT" %
%   B3:0/0  ALARM_SILENCE  "ALARM SILENCE PUSHBUTTON" %
% Rung: 520 %
SOR GRT N19:1 0 GRT F8:64 F18:0 XIO B3:0/1 BST TON T17:7 1.0 0 0 NXB XIC T17:7/DN OSR B3:33/3 OTE B3:33/4 BND EOR
%   N19:1  TT_7027_HIHI_DLY_SP  "TT-7027 HIHI ALARM DELAY SP FROM HMI" %
%   F8:64  TT_7027_SCI  "TT-7027 SCALED INPUT" %
%   F18:0  TT_7027_HIHI_SP  "TT-7027 HIHI ALARM SP" %
%   B3:0/1  ALARM_RESET  "ALARM RESET" %
%   T17:7  TT_7027_HIHI_DLY_TM  "TT-7027 HIHI ALARM DELAY" %
%   B3:33/3  "OSR" %
%   B3:33/4  "TT-7027 HIHI TRIGGER BIT" %
% Rung: 521 %
SOR BST BST XIC B3:33/4 NXB XIC B9:34/1 XIO B3:0/1 BND OTE B9:34/1 NXB BST XIC B3:33/4 NXB XIC B9:34/2 XIO B3:0/1 XIO B3:0/0 BND OTE B9:34/2 BND EOR
%   B3:33/4  "TT-7027 HIHI TRIGGER BIT" %
%   B9:34/1  TT_7027_HIHI_ALM  "TT-7027 HIHI ALARM BIT" %
%   B3:0/1  ALARM_RESET  "ALARM RESET" %
%   B9:34/2  TT_7027_HIHI_ALT  "TT-7027 HIHI ALERT BIT" %
%   B3:0/0  ALARM_SILENCE  "ALARM SILENCE PUSHBUTTON" %

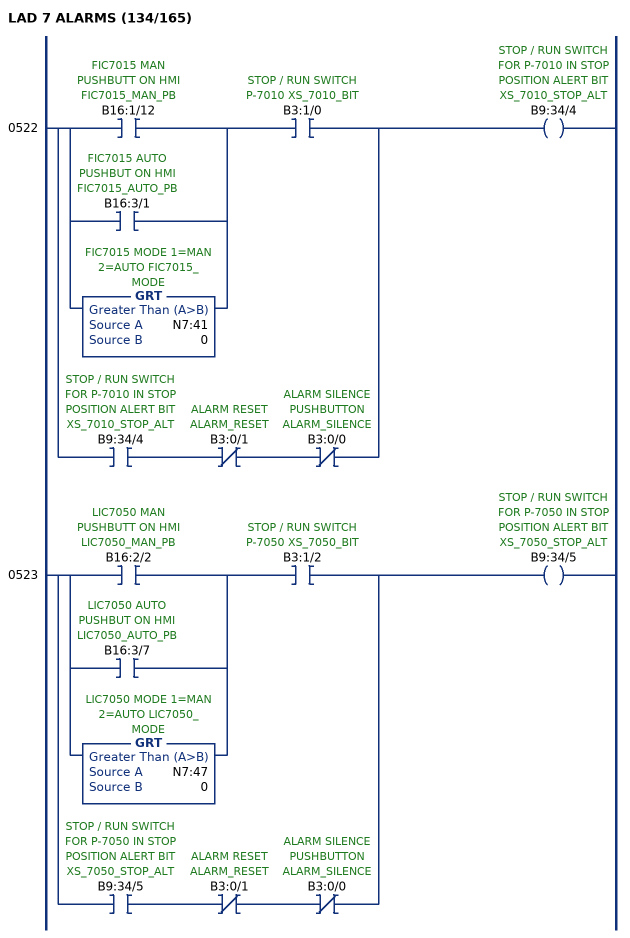
% Rung: 522 %
SOR BST BST XIC B16:1/12 NXB XIC B16:3/1 NXB GRT N7:41 0 BND XIC B3:1/0 NXB XIC B9:34/4 XIO B3:0/1 XIO B3:0/0 BND OTE B9:34/4 EOR
%   B16:1/12  FIC7015_MAN_PB  "FIC7015 MAN PUSHBUTT ON HMI" %
%   B16:3/1  FIC7015_AUTO_PB  "FIC7015 AUTO PUSHBUT ON HMI" %
%   N7:41  FIC7015_MODE  "FIC7015 MODE 1=MAN 2=AUTO" %
%   B3:1/0  XS_7010_BIT  "STOP / RUN SWITCH P-7010" %
%   B9:34/4  XS_7010_STOP_ALT  "STOP / RUN SWITCH FOR P-7010 IN STOP POSITION ALERT BIT" %
%   B3:0/1  ALARM_RESET  "ALARM RESET" %
%   B3:0/0  ALARM_SILENCE  "ALARM SILENCE PUSHBUTTON" %
% Rung: 523 %
SOR BST BST XIC B16:2/2 NXB XIC B16:3/7 NXB GRT N7:47 0 BND XIC B3:1/2 NXB XIC B9:34/5 XIO B3:0/1 XIO B3:0/0 BND OTE B9:34/5 EOR
%   B16:2/2  LIC7050_MAN_PB  "LIC7050 MAN PUSHBUTT ON HMI" %
%   B16:3/7  LIC7050_AUTO_PB  "LIC7050 AUTO PUSHBUT ON HMI" %
%   N7:47  LIC7050_MODE  "LIC7050 MODE 1=MAN 2=AUTO" %
%   B3:1/2  XS_7050_BIT  "STOP / RUN SWITCH P-7050" %
%   B9:34/5  XS_7050_STOP_ALT  "STOP / RUN SWITCH FOR P-7050 IN STOP POSITION ALERT BIT" %
%   B3:0/1  ALARM_RESET  "ALARM RESET" %
%   B3:0/0  ALARM_SILENCE  "ALARM SILENCE PUSHBUTTON" %

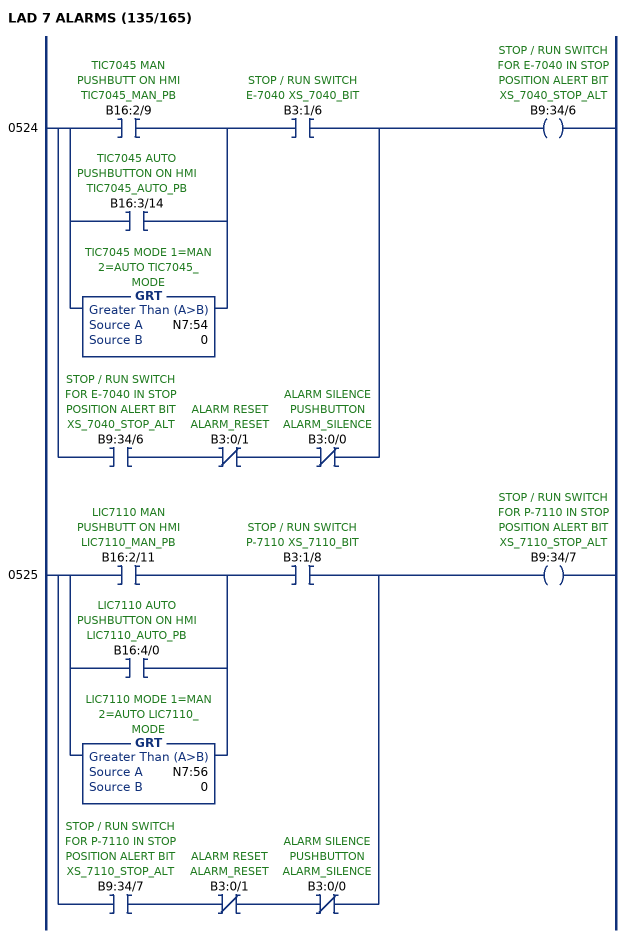
% Rung: 524 %
SOR BST BST XIC B16:2/9 NXB XIC B16:3/14 NXB GRT N7:54 0 BND XIC B3:1/6 NXB XIC B9:34/6 XIO B3:0/1 XIO B3:0/0 BND OTE B9:34/6 EOR
%   B16:2/9  TIC7045_MAN_PB  "TIC7045 MAN PUSHBUTT ON HMI" %
%   B16:3/14  TIC7045_AUTO_PB  "TIC7045 AUTO PUSHBUTTON ON HMI" %
%   N7:54  TIC7045_MODE  "TIC7045 MODE 1=MAN 2=AUTO" %
%   B3:1/6  XS_7040_BIT  "STOP / RUN SWITCH E-7040" %
%   B9:34/6  XS_7040_STOP_ALT  "STOP / RUN SWITCH FOR E-7040 IN STOP POSITION ALERT BIT" %
%   B3:0/1  ALARM_RESET  "ALARM RESET" %
%   B3:0/0  ALARM_SILENCE  "ALARM SILENCE PUSHBUTTON" %
% Rung: 525 %
SOR BST BST XIC B16:2/11 NXB XIC B16:4/0 NXB GRT N7:56 0 BND XIC B3:1/8 NXB XIC B9:34/7 XIO B3:0/1 XIO B3:0/0 BND OTE B9:34/7 EOR
%   B16:2/11  LIC7110_MAN_PB  "LIC7110 MAN PUSHBUTT ON HMI" %
%   B16:4/0  LIC7110_AUTO_PB  "LIC7110 AUTO PUSHBUTTON ON HMI" %
%   N7:56  LIC7110_MODE  "LIC7110 MODE 1=MAN 2=AUTO" %
%   B3:1/8  XS_7110_BIT  "STOP / RUN SWITCH P-7110" %
%   B9:34/7  XS_7110_STOP_ALT  "STOP / RUN SWITCH FOR P-7110 IN STOP POSITION ALERT BIT" %
%   B3:0/1  ALARM_RESET  "ALARM RESET" %
%   B3:0/0  ALARM_SILENCE  "ALARM SILENCE PUSHBUTTON" %

